(* PLC project EbN0扫描捕获_1度波束扫描及自跟踪优化 - 副本.project, CODESYS CODESYS V3.5 SP18 *)
(* stored: creationDateTime 2026-09-07T15:59:43.6480034, modificationDateTime 2026-09-07T15:13:02.4001786 *)

TYPE AxisCrtlStruct :
STRUCT
	iMode:INT;                     //方位运动模式   
	//bEnable :BOOL;                 //方位使能      
	rPosCmd :REAL;                 //方位位置命令    
	rVelCmd :REAL;                 //方位速度指令  
	rPIDCmdVel:LREAL;                //PID下发速度
	rPIDCmdPos:LREAL;				//PID目标位置
	bPIDEnable :BOOL;              //方位PID使能  
	bStartAutoTrack :BOOL;			//自跟踪使能
	rChanU:REAL;					//自跟踪采用的跟踪接收机误差电压
	
	rP:REAL:=1.0;                        //  P 
	rI:REAL:=0;                         //  I 
	rD:REAL:=0;                         //  D 
	rPIDThre:INT:=1;                   //积分阈值
	
	rP_AutoTrack:REAL:=3.0;          //自跟踪P
	rI_AutoTrack:REAL:=0.02;         //自跟踪I
	
	rAcceleration :REAL:=3;             //加速度
	rDeceleration :REAL:=3;       		//减速度
	rJogVel:LREAL:=2;					//点动速度 
	Pos_Vel:REAL:=4;					//位置模式速度
	rPos_Limit:LREAL;					//最大位置限制
	rVel_Limit:LREAL:=3;				//最大速度限制
	    
	rSoft_limit_Postive:REAL;
	rSoft_limit_Negative:REAL;			//正负软限位
	rLimitionNegative:LREAL;			//起始减速负限位
	rLimitionPositive:LREAL;			//起始减速正限位
	
END_STRUCT
END_TYPE

TYPE AxisStatus :
STRUCT
	Valid:BOOL;            //轴可用
	Busy:BOOL;             //轴工作中
	Error:BOOL;            //轴报错
	ErrorID:UINT;          //错误码
	ErrorStop:BOOL;        //轴错误停止
	Disabled:BOOL;         //轴下使能
	Stopping:BOOL;         //轴挂机或停止中
	Homing:BOOL;           //轴回原点
	Standstill:BOOL;       //轴待命
	DiscreteMotion:BOOL;   //轴离散运动
	ContinuousMotion:BOOL; //轴连续运动
	bServo_Enable:BOOL;		//轴使能状态
	bBrake:BOOL;			//轴抱闸状态
	Moving:BOOL;           //轴运动中
END_STRUCT
END_TYPE

TYPE AxisVisible :
STRUCT
	
	
	bJog_Forward:BOOL :=FALSE;
	bJog_Backward:BOOL :=FALSE;
	bVel_Run:BOOL:=FALSE;
	bPos_Run:BOOL:=FALSE;
	

	
	//JogB:BOOL;//点动指示灯
	//JogF:BOOL;
	bEnable:BOOL;//使能指示灯
	bUnable:BOOL;//下使能指示灯
	bLocalCtrl:BOOL;//本控指示灯
	bRemoteCtrl:BOOL;//远控指示灯
	//bJogLight:BOOL;//点动指示灯
	bStop:BOOL;//停止指示灯
	bmoveLight:BOOL;
	//bMovePos:BOOL;//速度运行指示灯
	//bMoveVel:BOOL;//位置运行指示灯
	bErrLight:BOOL;//报错提示灯
	//bExitPosLight:BOOL;//退限位模式指示灯
	//bPosLimLight:BOOL;//撞限位指示灯
	
	
	rLocalPosCmd:REAL;//本控位置命令
	rLocalVelCmd:REAL;//本控速度命令
	//rVelStep:REAL;//速度步距
	//rPosStep:REAL;//位置步距
END_STRUCT
END_TYPE

{attribute 'qualified_only'}
{attribute 'strict'}
TYPE MODES :
(
	powerOff:=0,          //下电
	powerOn := 1,         //上电
	positionMode:=2,      //位置模式
	velocityMode:=3,      //手动速度模式
	programBootMode:=4,   //程序引导模式
	reset:=6,             //轴错误复位
	halt:=7,              //停止
	stop:=8,             //挂机
	jog:=9 ,             //退限位模式
	edge:=10,            //
	test1:=11
);
END_TYPE

TYPE Word2Bit : UNION
  Apart_Word : WORD;
  Apart_Byte : ARRAY[1..2] OF BYTE;
  Apart_Real : REAL;  (* Apart_Bit:ARRAY[1..32]OF BIT; *)
  Apart_Int : INT;
END_UNION;
END_TYPE

TYPE Dword2Bit : UNION
  Apart_Dword : DWORD;
  Apart_Word : ARRAY[1..2] OF WORD;
  Apart_Byte : ARRAY[1..4] OF BYTE;
  Apart_Real : REAL;  (* Apart_Bit:ARRAY[1..32]OF BIT; *)
  Apart_Int : INT;
END_UNION;
END_TYPE

TYPE float2bit : UNION
  Apart_ulint : ULINT;
  Apart_dword : ARRAY[1..2] OF DWORD;
  Apart_word : ARRAY[1..4] OF WORD;
  Apart_byte : ARRAY[1..8] OF BYTE;
  Apart_real : ARRAY[1..2] OF REAL;  (* Apart_bit:ARRAY[1..64]OF Util.BIT_AS_DWORD; *)
  Apart_int : ARRAY[1..4] OF INT;
END_UNION;
END_TYPE

TYPE UnionLREAL_WORD : UNION
  lrealValue : LREAL;
  words : ARRAY[1..4] OF WORD;
END_UNION;
END_TYPE

TYPE Time2Word : UNION
  uliData : ULINT;
  wWords : ARRAY[1..4] OF WORD;
  lrReal : LREAL;
  arReal : ARRAY[0..1] OF REAL;
END_UNION;
END_TYPE

PROGRAM PLC_PRG
VAR
	a : DINT;
	b : REAL;
END_VAR

                    a := REAL_TO_DINT(b * 524288 / 360);
                  
END_PROGRAM

PROGRAM TimeCase
VAR
	stUTC_Timestamp :SYSTIME ;
	stSYS_Timestamp :ULINT ;
	stGNSS_Timestap :ULINT;
    Result : RTS_IEC_RESULT;
	Uptriger:Standard.R_TRIG;
	Triger AT %IX0.0:BOOL;
	Feed AT %QX0.0:BOOL;	
	TON_F: TON;
	dDelPTime: DINT;
	max_DelPTime:DINT :=0; 
	min_DelPTime: DINT :=-999999;
	iCount: INT;
	dtNow: DATE_AND_TIME;
	dtGNSS: DATE_AND_TIME;
	dtLastGNSS: ULINT;
	iDiffETime: DINT;
	DelPTime: DINT;
	
END_VAR

                    //计算时间误差序列
Result := SysTimeRtcHighResGet(stUTC_Timestamp);        
stSYS_Timestamp := TO_ULINT(stUTC_Timestamp);           // ULINT，获取本地时间
dtNow := TO_DT(stUTC_Timestamp / 1000); 		        // 转换为DATE_AND_TIME类型

Uptriger(CLK:=Triger);                                  //检测PPS上升沿
IF Uptriger.Q THEN                                      //上升沿触发后，GPRMC解析，DO0上升沿输出（电平24V）
	Feed:=TRUE;	
	dtGNSS := TO_DT(GVL.stGNSS_Timestap / 1000); 	    // 拿到串口时间数据			                                     
	iDiffETime:=ULINT_TO_DINT(GVL.stGNSS_Timestap-dtLastGNSS);  
	dtLastGNSS:=GVL.stGNSS_Timestap;                    //缓存上一周期时间戳（ms)  
	dDelPTime:=ULINT_TO_DINT(GVL.stGNSS_Timestap - stSYS_Timestamp);       //计算误差	              
	IF iDiffETime = 1000 THEN                           //确保时间更新步进1S
		IF dDelPTime < 0 THEN                           //更新最小值
			IF dDelPTime < min_DelPTime THEN
				min_DelPTime:=dDelPTime;
				DelPTime:=min_DelPTime;                 
			END_IF		
		ELSE                                            //更新最大值
			IF dDelPTime > max_DelPTime THEN
				max_DelPTime:=dDelPTime;
				DelPTime:=max_DelPTime;
			END_IF
		END_IF	
	END_IF				    						
	iCount:=iCount+1;
	IF iCount >= 60 THEN                                //一分钟校一次时间
		GVL.dDelTime:=DelPTime;
		max_DelPTime:=0;
		min_DelPTime:=0;	
		iCount:=0;
	END_IF
	
END_IF
TON_F(IN:=Feed, PT:=T#100MS, Q=>,ET=>);                 //脉宽200ms（测试时延，为了在示波器看波形）
IF TON_F.Q THEN
	Feed:=FALSE;		
END_IF
                  
END_PROGRAM

FUNCTION_BLOCK PID
VAR_INPUT
    rTarget : REAL;       (* 设定值 *)
    rFeedback : REAL;       (* 反馈值 *)
	rPosLimPositive:LREAL;//位置正限位
	rPosLimNegative:LREAL;//位置反限位
	rKp:REAL;     //比例增益
	rKi:REAL;     //积分增益
	rKd:REAL;     //微分增益
	iThreshold:INT;//积分项开启的位置阈值
	bPIDEnable:BOOL:=TRUE;//PID使能
	rVelLim:LREAL;//速度限制
END_VAR
VAR_OUTPUT
    rPIDOutput : LREAL:=0;         //带方向的输出速度
	rPIDtrace : LREAL:=0;         //带方向的输出速度
END_VAR
VAR
	//rPIDOutPut: REAL:=0.0;
	rLastError: LREAL:=0.0;(*上一次误差*)
	rErrorNow:LREAL:=0.0;(*当前误差*)
    rIntegralNew : LREAL := 0.0; (* 积分项 *)
    rDerivativeNew : LREAL := 0.0; (* 微分项 *)
	rDelta: LREAL;(*增量*)
	rProportionNew: LREAL;
	
	//iAzPIDEnable: INT;
END_VAR

                    
IF (bPIDEnable>0) THEN //如果PID使能
	IF rTarget=rFeedback THEN
		rPIDOutput:=0;	
	ELSE
	
		rErrorNow:=rTarget-rFeedback;//计算当前误差 en
		rProportionNew:=rErrorNow;//比例项
		//积分项
		IF rFeedback>rPosLimNegative AND rFeedback<rPosLimPositive THEN //若在软限位之内，工作时开启积分项
			IF (ABS(rTarget-rFeedback)<iThreshold) THEN//位置差小于积分阈值
				rIntegralNew:= rIntegralNew+rErrorNow; //积分项
			ELSE
				rIntegralNew:=0;
			END_IF;
		ELSE //不在软限位范围内,则积分项为0
			rIntegralNew:=0;
		END_IF

		//PID输出
		rPIDOutPut:=rKp*rProportionNew+rKi*rIntegralNew;
		rPIDtrace:=rKp*rProportionNew+rKi*rIntegralNew;


		//PID限速
		
			IF rPIDOutput<(-rVelLim) THEN
				rPIDOutput:=-rVelLim;
			ELSIF rPIDOutput>rVelLim THEN
				rPIDOutput:=rVelLim;
			END_IF
		
		
		IF rFeedback>rPosLimPositive AND rPIDOutput>0 THEN 
			rPIDOutput:=0;
		END_IF
		IF rFeedback<rPosLimNegative AND rPIDOutput<0 THEN
			rPIDOutput:=0;
		END_IF
		
		rLastError:=rErrorNow;//将当前误差赋值给上一次误差
		
	END_IF
ELSE//非使能清零PID各项
	rProportionNew:=0.0;
	rIntegralNew:=0.0;
	rPIDOutput:=0.0;
END_IF










                  
END_FUNCTION_BLOCK

PROGRAM TimeAdd
VAR
	icount : INT;
	iSecondLast:INT;
END_VAR

                    // 监测时统串口状态，时间插值
IF iSecondLast <> GPRMC_1.iSecond THEN
	icount := 0;
ELSE
	icount := icount + 1;
END_IF
iSecondLast := GPRMC_1.iSecond;

IF icount > 2000 THEN
	icount := 0;
END_IF
                  
END_PROGRAM

PROGRAM GPRMC
VAR
	com_init:gcan.FB_Com_Init;      		//gcan.FB_Com_Init为串口初始化功能块，可设定串口端口号，串口波特率等参数
	com_read:gcan.FB_Com_Read ;				//gcan.FB_Com_Read为串口接收功能块，用于通过接收串口发送给PLC的数据
	com_write:gcan.FB_Com_Write ;			//gcan.FB_Com_Write为串口发送功能块，用于发送串口数据
	m_uiError:UINT;							//用于承接功能块中报错引脚错误信息的变量
	m_out:BOOL;								//用于承接功能块中完成标志引脚数据的变量
	isFirst:BOOL:=TRUE;						//用于判断初始化只执行一次的逻辑
	mPort:BYTE;								//程序中用作设定串口端口号
	recSize:UINT;							//接收数据长度，单位：字节
	recBuf:ARRAY[0..100] OF BYTE;			//用于存放接收到的串口数据的数组
	sum_i:INT;
	checksum:BYTE;
	iYear: INT;
	iMonth: INT;
	iDay: INT;
	iHour: INT;
	iMinute: INT;
	iSecond: INT;
	strDateTimeNow : STRING;
	gnssTimestamp: ULINT;
	high4: BYTE;
	low4: BYTE;
END_VAR

                    ////////////////////////////////////////////////////////////////////////////////////////
//串口接收GPRMC报文解析
//日期：2024/08/25
//版本：V1.1
/////////////////////////////////////////////////////////////////////////////////////////

mPort:=1;								//串口端口号设定，GCAN-PLC-400、GCAN-PLC-510、GCAN-PLC-511，1为232，2为485
										//GCAN-PLC-324、GCAN-PLC-326，1为第一路485，2为第2路485
IF isFirst THEN
	com_init(							//串口初始化功能块
	EN_IN:=TRUE,						//串口初始化功能块使能
	xEnable:=TRUE,						//串口功能使能
	bPort:=mPort,						//串口端口号设定
	uiBaudrate:=115200,					//串口波特率设定
	bParity:=0,							//串口奇偶校验设定，0为无校验，1为奇校验，2为偶检验
	bDatabits:=8,						//数据位设定
	bStopbits:=1,						//停止位设定
	EN_OUT=>m_out,						//串口初始化功能块执行完成标志位
	uiError=>m_uiError);				//串口初始化功能块执行错误信息
	isfirst:=FALSE;						//执行一次初始化后关闭IF的条件使其之后进入ELSE程序段运行

ELSE
	
		com_read(						//串口读取功能块
		EN_in:=TRUE,					//读取功能块使能，为TRUE执行读取
		bPort:=mPort,					//串口端口号设定
		p_brxdata:=ADR(recBuf),			//读取到的串口数据引脚为指针类型，使用ADR()指向自建数组将数据存放到数组中
		uiMaxsize:=100,					//设定最大读取长度
		EN_out=>m_out,					//串口读取功能块执行完成标志位******功能块执行完成不代表接收完成********
		uiRecSize=>recSize,				//串口接收数据长度，单位：字节，大于0时说明接收到数据可用于判断是否接收
		uierror=>m_uierror);			//串口读取功能块执行错误信息
										//从数组recBuf里取数据，解析出年、月、日、时、分、秒
		//有效判定(A)+和校验(hh),前 4bit和后 4bit的 16 进制数分别以 ASCII 码表示(0~9,A~F)，高位在前。
		IF 	recBuf[17] = 65 THEN
(*			checksum := 16#00;
			FOR sum_i:=1 TO 74 BY 1 DO
				checksum:= checksum XOR recBuf[sum_i];
			END_FOR
			high4 := (SHR(checksum, 4) AND 16#0F)+16#30;
			low4 := (checksum AND 16#0F)+16#30;
			IF recBuf[76]= high4 AND recBuf[77]= low4 THEN 
*)			IF recBuf[60] = 44 THEN // 航向角 x.x
				iYear:=BYTE_TO_INT(recBuf[65]-48)*10+BYTE_TO_INT(recBuf[66]-48)+2000;
				iMonth:=BYTE_TO_INT(recBuf[63]-48)*10+BYTE_TO_INT(recBuf[64]-48);
				iDay:=BYTE_TO_INT(recBuf[61]-48)*10+BYTE_TO_INT(recBuf[62]-48);
				iHour:=BYTE_TO_INT(recBuf[7]-48)*10+BYTE_TO_INT(recBuf[8]-48)+8;
				iMinute:=BYTE_TO_INT(recBuf[9]-48)*10+BYTE_TO_INT(recBuf[10]-48);
				iSecond:=BYTE_TO_INT(recBuf[11]-48)*10+BYTE_TO_INT(recBuf[12]-48);
			END_IF
			IF recBuf[61] = 44 THEN // 航向角 xx.x
				iYear:=BYTE_TO_INT(recBuf[66]-48)*10+BYTE_TO_INT(recBuf[67]-48)+2000;
				iMonth:=BYTE_TO_INT(recBuf[64]-48)*10+BYTE_TO_INT(recBuf[65]-48);
				iDay:=BYTE_TO_INT(recBuf[62]-48)*10+BYTE_TO_INT(recBuf[63]-48);
				iHour:=BYTE_TO_INT(recBuf[7]-48)*10+BYTE_TO_INT(recBuf[8]-48)+8;
				iMinute:=BYTE_TO_INT(recBuf[9]-48)*10+BYTE_TO_INT(recBuf[10]-48);
				iSecond:=BYTE_TO_INT(recBuf[11]-48)*10+BYTE_TO_INT(recBuf[12]-48);
			END_IF
			IF recBuf[62] = 44 THEN // 航向角 xxx.x
				iYear:=BYTE_TO_INT(recBuf[67]-48)*10+BYTE_TO_INT(recBuf[68]-48)+2000;
				iMonth:=BYTE_TO_INT(recBuf[65]-48)*10+BYTE_TO_INT(recBuf[66]-48);
				iDay:=BYTE_TO_INT(recBuf[63]-48)*10+BYTE_TO_INT(recBuf[64]-48);
				iHour:=BYTE_TO_INT(recBuf[7]-48)*10+BYTE_TO_INT(recBuf[8]-48)+8;
				iMinute:=BYTE_TO_INT(recBuf[9]-48)*10+BYTE_TO_INT(recBuf[10]-48);
				iSecond:=BYTE_TO_INT(recBuf[11]-48)*10+BYTE_TO_INT(recBuf[12]-48);
			END_IF
				// 计算时间戳		
				strDateTimeNow := CONCAT(STR1 := 'DT#', STR2 := INT_TO_STRING(iYear));
				strDateTimeNow := CONCAT(STR1 := strDateTimeNow, STR2 := '-');
				strDateTimeNow := CONCAT(STR1 := strDateTimeNow, STR2 := INT_TO_STRING(iMonth));
				strDateTimeNow := CONCAT(STR1 := strDateTimeNow, STR2 := '-');
				strDateTimeNow := CONCAT(STR1 := strDateTimeNow, STR2 := INT_TO_STRING(iDay));
				strDateTimeNow := CONCAT(STR1 := strDateTimeNow, STR2 := '-');
				strDateTimeNow := CONCAT(STR1 := strDateTimeNow, STR2 := INT_TO_STRING(iHour));
				strDateTimeNow := CONCAT(STR1 := strDateTimeNow, STR2 := ':');
				strDateTimeNow := CONCAT(STR1 := strDateTimeNow, STR2 := INT_TO_STRING(iMinute));
				strDateTimeNow := CONCAT(STR1 := strDateTimeNow, STR2 := ':');
				strDateTimeNow := CONCAT(STR1 := strDateTimeNow, STR2 := INT_TO_STRING(iSecond));
				gnssTimestamp := DT_TO_ULINT(TO_DT(strDateTimeNow)) * 1000;
				GVL.stGNSS_Timestap := gnssTimestamp;
			//END_IF
		END_IF
					


(*	IF recsize>0 THEN					//如果接收到串口数据
		
		com_write(						//串口发送功能块
		EN_IN:=TRUE,					//串口发送功能块使能，发送机制：当使能为TRUE时，PLC程序每周期运行到此处就执行一次发送
		bPort:=mPort,					//串口端口号设定
		p_bTxdata:=ADR(recbuf),			//将接收存放到数组中的数据发送出去******若发送其它数据，自建另一数组用于存放发送数据即可
		uiTxsize:=recsize,				//发送长度为接收到的数据长度******若发送其它长度，自行填写所需长度即可
		EN_OUT=>m_out,					//串口发送功能块执行完成标志位
		uierror=>m_uierror);			//串口发送功能块执行错误信息
			
	END_IF
*)	
END_IF
                  
END_PROGRAM

PROGRAM RealTimePosCal
VAR
	dtReal: DATE_AND_TIME;
	sRealTime:STRING;
	btestTimeInit:BOOL;
	AzCubicInter:threesimple2_1;//方位三次样条插值
	ElCubicInter:threesimple2_1;//俯仰三次样条插值
	iErrcode : INT;
	rInterAzPos:REAL;//方位轴插值位置
    rInterElPos:REAL;//俯仰轴插值位置
	
	rInterAzPostest:REAL;//方位轴插值位置
    rInterElPostest:REAL;//俯仰轴插值位置
	
	rPolyAzPos:REAL;//方位轴多项式位置
    rPolyElPos:REAL;//俯仰轴多项式位置
	AzPoly:Get_AZ;
	ElPoly:Get_AZ_1;
	
	dRTime:ULINT;//上位机外部时间 单位ns Unix时间戳，起点是1970-1-1 0:0:0
	dLastRTime:ULINT;
	icount : INT;
END_VAR

                    //GVL.dRealTime:= TimeCase.stSYS_Timestamp + GVL.dDelTime + 1000 + 56 ;// 矫正后的时间 单位毫秒
//GVL.dRealTime:= TimeCase.stSYS_Timestamp + GVL.dDelTime;// 矫正后的时间 单位毫秒

//直接从上位机拿数
dRTime := modbus_slave.UTC_New + 8 * 3600 * 1000;
IF dRTime <> dLastRTime THEN
	icount := 0;
ELSE 
	icount := icount + 1;
END_IF
dLastRTime:=dRTime;
IF not GVL.bTimeSwich THEN
	GVL.dRealTime:=GVL.stGNSS_Timestap + 10*timeadd.icount;
ELSE
	GVL.dRealTime:=dRTime + 10*icount;
END_IF
IF icount > 5000 THEN
	icount := 0;
END_IF
(*
GVL.dRealTime:=GVL.stGNSS_Timestap + 10*timeadd.icount;
*)
dtReal := TO_DT(GVL.dRealTime / 1000);
sRealTime := TO_STRING(dtReal);

IF Axis1Remote.iMode=4 AND Axis2Remote.iMode=4 THEN//若PTP时间锁定 且时间模式为PTP时间
		//三次样条插值

		//GVL.dRealTime:= TimeCase.stSYS_Timestamp + GVL.dDelTime + 1000 + 56; // 矫正后的时间 单位毫秒
		IF NOT GVL.bTimeSwich THEN
			GVL.dRealTime:=GVL.stGNSS_Timestap + 10*timeadd.icount;
		ELSE
			GVL.dRealTime:=dRTime + 10*icount;
		END_IF
		AzCubicInter(XModbusUL:=Modbus_Slave.aUTC_TIME,YModbus:=Modbus_Slave.aPosCmd_2,y0:=0,yn:=0,xt:=(ULINT_TO_LREAL(GVL.dRealTime) - 8 * 3600 *1000),sout=>rInterAzPos,ErrCode=>iErrcode);
		ElCubicInter(XModbusUL:=Modbus_Slave.aUTC_TIME,YModbus:=Modbus_Slave.aPosCmd_1,y0:=0,yn:=0,xt:=(ULINT_TO_LREAL(GVL.dRealTime) - 8 * 3600 *1000),sout=>rInterElPos,ErrCode=>iErrcode);
		IF iErrcode>0 THEN //模块内错误代码清0 外部维持
			Error_code:=iErrcode;
		END_IF
END_IF
(*
//IF Axis1Remote.iMode=4 AND Axis2Remote.iMode=4 AND Modbus_Slave.bIFPoly THEN//若PTP时间锁定 且时间模式为PTP时间
IF Modbus_Slave.bIFPoly THEN//若PTP时间锁定 且时间模式为PTP时间
		//多项式拟合

		//GVL.dRealTime:= TimeCase.stSYS_Timestamp + GVL.dDelTime + 1000 + 56; // 矫正后的时间 单位毫秒
		GVL.dRealTime:= GVL.stGNSS_Timestap +450; // 矫正后的时间 单位毫秒
	
		AzPoly(
		uliRealTime := (ULINT_TO_LREAL(GVL.dRealTime) - 8 * 3600 *1000),
		lrStartTime := Modbus_Slave.starttime,
		rNodeTime1 := Modbus_Slave.rNodeTime1_az,
		rNodeTime2 := Modbus_Slave.rNodeTime2_az,
		rNodeTime3 := Modbus_Slave.rNodeTime3_az,
		rNodeTime4 := Modbus_Slave.rNodeTime4_az,
		rNodeTime5 := Modbus_Slave.rNodeTime5_az,
		rEndTime := Modbus_Slave.rEndTime,
		lrFun1 := Modbus_Slave.lrFun1_az,
		lrFun2 := Modbus_Slave.lrFun2_az,
		lrFun3 := Modbus_Slave.lrFun3_az,
		lrFun4 := Modbus_Slave.lrFun4_az,
		lrFun5 := Modbus_Slave.lrFun5_az,
		lrFun6 := Modbus_Slave.lrFun6_az,
		lrFitResult => rPolyAzPos);
		
		ElPoly(
		uliRealTime := (ULINT_TO_LREAL(GVL.dRealTime) - 8 * 3600 *1000),
		lrStartTime := Modbus_Slave.starttime,
		rNodeTime1 := Modbus_Slave.rNodeTime1_el,
		rNodeTime2 := Modbus_Slave.rNodeTime2_el,
		rNodeTime3 := Modbus_Slave.rNodeTime3_el,
		rNodeTime4 := Modbus_Slave.rNodeTime4_el,
		rNodeTime5 := Modbus_Slave.rNodeTime5_el,
		rEndTime := Modbus_Slave.rEndTime,
		lrFun1 := Modbus_Slave.lrFun1_el,
		lrFun2 := Modbus_Slave.lrFun2_el,
		lrFun3 := Modbus_Slave.lrFun3_el,
		lrFun4 := Modbus_Slave.lrFun4_el,
		lrFun5 := Modbus_Slave.lrFun5_el,
		lrFun6 := Modbus_Slave.lrFun6_el,
		lrFitResult => rPolyElPos);
		
		rInterAzPos := rPolyAzPos * (-1);
		rInterElPos := rPolyElPos + 90;
END_IF
*)
                  
END_PROGRAM

PROGRAM Modbus_Slave
VAR
	modTcpSlaveInit:gcan.FB_ModbusTCP_Slave_Init;	//gcan.FB_ModbusTCP_Slave_Init为Modbus TCP Slave初始化功能块
	modTcpSlaveCtrl:gcan.FB_ModbusTCP_Slave_Ctrl;	//gcan.FB_ModbusTCP_Slave_Init为Modbus TCP Slave执行功能块
	eout: BOOL;										//用于承接功能块中完成标志引脚数据的变量
	iSocket: INT;									//用于存放自身socket
	uiErr: UINT;									//用于承接功能块中报错引脚错误信息的变量
	isInit: BOOL:=FALSE;							//用于初始化执行一次的逻辑变量
	arClient:ARRAY[0..10] OF INT;					//用于存放Client即主站的socket
	
	arDo_data:ARRAY[0..654] OF BOOL;					//用于存放线圈的数据
	arDi_data:ARRAY[0..79] OF BOOL;					//用于存放离散型数据
	//arReg_data:ARRAY[0..10] OF INT;					//用于存放保持型寄存器的数据
	//arAi_data:ARRAY[0..10] OF INT;					//用于存放输入型寄存器的数据
	modbusData	    AT %MW0		: ARRAY[0..654] OF WORD;//用于存放保持型寄存器的数据，接收的数据
	modbusInputRegs	AT %MW660	: ARRAY[0..79] OF WORD;//用于存放输入型寄存器的数据，上报的数据
	
	enCtr:BOOL:=FALSE;								//Modbus TCP Slave执行功能块使能变量

	Remote_time 	 	:LWORD;
	dif:ULINT;//时延
	iCount				:WORD;
	TypeList1 			:DWORD;
	UTC_Union: float2bit;
	CtrlBool: WORD_AS_BIT;
	bCommReset:BOOL;		//错误复位标识符
	iWatchDogTime:INT;
	
	Pos1_Union:float2bit;//远控处理数据结构体
	Pos2_Union:float2bit;
	Pos3_Union:float2bit;
	//轴1远控指令，俯仰
	iMode_1 			:INT;  			//轴1模式远控
	rPosCmd_1 		 	:REAL; 			//轴1位置指令远控
	rVelcmd_1 			:REAL; 			//轴1速度指令远控
	rP_1 				:REAL;    	//轴1P远控
	rI_1 			 	:REAL;      	//轴1I远控
	rD_1				:REAL;     	//轴1D远控
	rThreshold_1 	 	:INT:=1;		//轴1积分阈值远控
	rAcceleration_1  	:REAL;			//最大加速度
	rDeceleration_1  	:REAL;			//最大减速度	
	rVelLim_1	  	 	:REAL;			//最大速度
	
	//轴2远控指令，方位
    iMode_2  		 	:INT; 			//轴2模式远控
	rPosCmd_2 			:REAL; 			//轴2位置指令远控
	rVelcmd_2 			:REAL; 			//轴2速度指令远控
	rP_2 				:REAL;  		//轴2P远控
	rI_2 			 	:REAL;  		//轴2I远控
	rD_2 			 	:REAL;  		//轴2D远控
	rThreshold_2 		:INT;			//轴2积分阈值远控
	rAcceleration_2 	:REAL;			//最大加速度
	rDeceleration_2  	:REAL;			//最大减速度	
	rVelLim_2	  		:REAL;			//最大速度
	//轴3远控指令，方位
    iMode_3  		 	:INT; 			//轴2模式远控
	rPosCmd_3 			:REAL; 			//轴2位置指令远控
	rVelcmd_3 			:REAL; 			//轴2速度指令远控
	rP_3 				:REAL;  		//轴2P远控
	rI_3 			 	:REAL;  		//轴2I远控
	rD_3 			 	:REAL;  		//轴2D远控
	rThreshold_3 		:INT;			//轴2积分阈值远控
	rAcceleration_3 	:REAL;			//最大加速度
	rDeceleration_3  	:REAL;			//最大减速度	
	rVelLim_3	  		:REAL;			//最大速度
	
	//轨道时间结构体
	UTC_Orbit_Union:float2bit;
	UTC_Orbit_New:ULINT;
	UTC_Orbit_Last:ULINT;
	//拉偏变量
	TimeBias_Union:float2bit;
	Bias1_Union:float2bit;
	Bias2_Union:float2bit;
	Bias3_Union:float2bit;
	AcuElOffset:float2bit;
	rTimeBias:LREAL;
	rBias_1:LREAL;
	rBias_2:LREAL;
	rBias_3:LREAL;
	lrElOffset:LREAL;
	UTC_New:ULINT;
	UTC_Last:ULINT;
	aUTC_TIME:ARRAY [1..10] OF ULINT;  //用于三次样条插值的数据
	aPosCmd_1 :ARRAY [1..10] OF LREAL;//用于三次样条插值的数据
	aPosCmd_2 :ARRAY [1..10] OF LREAL;//用于三次样条插值的数据
	isave:INT;
	iCheck:INT;
	bPass:BOOL;//通过大小检测
	iclear:INT;
	
	uPTPTime_Union:float2bit;
	DI1_Union:Util.BIT_AS_WORD;	//上报位置结构体
	DI2_Union:Util.BIT_AS_WORD;
	DO1_Union:Util.BIT_AS_WORD;
	DO2_Union:Util.BIT_AS_WORD;
	DI1_word:WORD;
	DI2_word:WORD;
	DO1_word:WORD;
	DO2_word:WORD;
// 	
	PosSub1_Union:float2bit;
	PosSub2_Union:float2bit;
	PosSub3_Union:float2bit;
	BiasSub1_Union:float2bit;
	BiasSub2_Union:float2bit;
	BiasSub3_Union:float2bit;

	Chan_Union:Util.BIT_AS_WORD;
	Chan_word:WORD;
	
	ptptime:ULINT;
	
	rAzTheory:LREAL;
	rEltheory:LREAL;
	rAzTheory_Union:float2bit;
	rEltheory_Union:float2bit;
	
	
	MillisecondsTime: ULINT;
	
	// for time test
	DeltaTimeBetPC : ULINT;

	AGC_Value: REAL;

	// 方位轨道多项式变量
	starttime : LREAL ;
	rNodeTime1_az : LREAL;
	rNodeTime2_az : LREAL;
	rNodeTime3_az : LREAL;
    rNodeTime4_az : LREAL;
    rNodeTime5_az : LREAL;
	rEndTime : LREAL;
	
	lrFun1_az : ARRAY[0..10] OF LREAL;
    lrFun2_az : ARRAY[0..10] OF LREAL;
    lrFun3_az : ARRAY[0..10] OF LREAL;
    lrFun4_az : ARRAY[0..10] OF LREAL;
	lrFun5_az : ARRAY[0..10] OF LREAL;
    lrFun6_az : ARRAY[0..10] OF LREAL;

    unionFun1_az : ARRAY[0..10] OF UnionLREAL_WORD;
    unionFun2_az : ARRAY[0..10] OF UnionLREAL_WORD;
    unionFun3_az : ARRAY[0..10] OF UnionLREAL_WORD;
    unionFun4_az : ARRAY[0..10] OF UnionLREAL_WORD;
    unionFun5_az : ARRAY[0..10] OF UnionLREAL_WORD;
    unionFun6_az : ARRAY[0..10] OF UnionLREAL_WORD;
	
	unionStartTime: UnionLREAL_WORD;
	
    unionNodeTime1_az : UnionLREAL_WORD;
    unionNodeTime2_az : UnionLREAL_WORD;
    unionNodeTime3_az : UnionLREAL_WORD;
    unionNodeTime4_az : UnionLREAL_WORD;
    unionNodeTime5_az : UnionLREAL_WORD;
    unionEndTime : UnionLREAL_WORD;
	
	// 俯仰轨道多项式变量
	rNodeTime1_el : REAL;
	rNodeTime2_el : REAL;
	rNodeTime3_el : REAL;
    rNodeTime4_el : REAL;
    rNodeTime5_el : REAL;
	lrFun1_el : ARRAY[0..10] OF LREAL;
    lrFun2_el : ARRAY[0..10] OF LREAL;
    lrFun3_el : ARRAY[0..10] OF LREAL;
    lrFun4_el : ARRAY[0..10] OF LREAL;
	lrFun5_el : ARRAY[0..10] OF LREAL;
    lrFun6_el : ARRAY[0..10] OF LREAL;
	unionFun1_el : ARRAY[0..10] OF UnionLREAL_WORD;
	unionFun2_el : ARRAY[0..10] OF UnionLREAL_WORD;
	unionFun3_el : ARRAY[0..10] OF UnionLREAL_WORD;
	unionFun4_el : ARRAY[0..10] OF UnionLREAL_WORD;
	unionFun5_el : ARRAY[0..10] OF UnionLREAL_WORD;
	unionFun6_el : ARRAY[0..10] OF UnionLREAL_WORD;
	unionNodeTime1_el : UnionLREAL_WORD;
	unionNodeTime2_el : UnionLREAL_WORD;
	unionNodeTime3_el : UnionLREAL_WORD;
	unionNodeTime4_el : UnionLREAL_WORD;
	unionNodeTime5_el : UnionLREAL_WORD;
	unionSum:UnionLREAL_WORD;
	lrSum:LREAL;
	lrSumlocal:LREAL;
	i : INT;
	bNotFirst : BOOL; //
	bCheck : BOOL;
	bIFPoly: BOOL;//开启多项式拟合模式的标识，由上位机下发
	iCountPolyGet:INT;//计时接收多项式数组的模块
	uChangeTest:Time2Word;//变量转换测试
	iCountSum:INT;
	bSearch: BOOL;
	bStartTrackAcu : BOOL;
	
	//接收上位机下发位置模式速度
	rAzPosVel : REAL := 8;
	rElPosVel : REAL := 6;
	rTlPosVel : REAL := 8;
END_VAR

                    IF isInit=FALSE THEN							
	
	modtcpslaveinit(en_in:=TRUE,					//Modbus TCP Slave初始化功能块使能
	xenable:=TRUE,									//使能初始化功能
	iport:=502,										//开放端口号502
	en_out=>eout,									//Modbus TCP Slave初始化功能块执行完成
	isocket=>iSocket,								//创建的socket存入变量
	uierror=>uiErr);								//Modbus TCP Slave初始化功能块执行错误信息
	
	IF isocket>=0 AND uiErr=0 THEN					//成功创建socket且无错误，逻辑标志置位，下周期执行ELSE
		isInit:=TRUE;	
		
		enCtr:=FALSE;
		ELSE                                        //等待连接成功
		modtcpslaveinit(en_in:=0,xenable:=0);	
	END_IF
	
 
ELSE
	
	modtcpslavectrl(en_in:=enCtr,					//Modbus TCP Slave执行功能块使能
	xenable:=TRUE,									//Modbus TCP Slave执行功能使能
	isocket:=isocket,								//输入创建的socket
	dwatchdogtime:=2000,							//看门狗时间
	p_clientsocket:=ADR(arClient),					//将连接进来的socket存放到数组
	imaxclientcount:=10,							//设置最大连接数量
	uido_number:=10,uido_startaddr:=0,pdo_data:=ADR(ardo_data),		//uido_number设定线圈个数，uido_startaddr设定线圈起始地址，数据存放在ardo_data数组
	uidi_number:=10,uidi_startaddr:=0,pdi_data:=ADR(ardi_data),		//uidi_number设定离散型数据个数，uidi_startaddr设定离散型数据起始地址，数据存放在ardi_data数组
	uireg_number:=655,uireg_startaddr:=0,preg_data:=ADR(modbusData), //uireg_number设定保持型寄存器个数，uireg_startaddr设定保持型寄存器起始地址，数据存放在arreg_data数组
	uiai_number:=79,uiai_startaddr:=0,pai_data:=ADR(modbusInputRegs),//uiai_number设定输入型寄存器个数，uiai_startaddr设定输入型寄存器起始地址，数据存放在arai_data数组
	en_out=>eout,									//Modbus TCP Slave执行功能块执行完成
	uierror=>uierr);								//Modbus TCP Slave执行功能块执行错误信息
	enctr:=TRUE;
	IF uierr <>0 THEN                               //如果从站报错，则重新连接从站
		modtcpslaveinit(en_in:=0,xenable:=0);	
		isInit:=0;
	END_IF
	//iMode:  0 下电  1 上电  2 速度模式  3 停止  4 位置模式  5 继续运行
	//方位轴指令
(*
	Az_ctrl.iMode:=WORD_TO_INT(modbusData[0]);
	AZ_ctrl.rTarVel:=WORD_TO_REAL(modbusData[1]);
	AZ_ctrl.rTarPos:=WORD_TO_REAL(modbusData[2])*-1.0;
	
	//俯仰轴指令
	El_ctrl.iMode:=WORD_TO_INT(modbusData[10]);
	El_ctrl.rTarVel:=WORD_TO_REAL(modbusData[11]);
	El_ctrl.rTarPos:=WORD_TO_REAL(modbusData[12])+90.0;
	*)
	
	// modbus下发数据
	UTC_Union.Apart_word[1]:=modbusData[3];
	UTC_Union.Apart_word[2]:=modbusData[2];
	UTC_Union.Apart_word[3]:=modbusData[1];
	UTC_Union.Apart_word[4]:=modbusData[0];
	UTC_New:=UTC_Union.Apart_ulint;
	DeltaTimeBetPC := UTC_New - TO_ULINT(GVL.dRealTime);
	CtrlBool(W:=modbusData[7],
			B14=>bCommReset,
			B13=>Axis2Remote.bPIDEnable,
			B12=>Axis1Remote.bPIDEnable,
			B11=>Axis3Remote.bPIDEnable,
			B10=>bStartTrackAcu,
			B07=>bIFPoly,
			B06=>bSearch, //十字搜索开启标识
			);
	//方位轴指令
	iMode_2:=WORD_TO_INT(modbusData[8]);
	Pos2_Union.Apart_word[2]:=modbusData[9];
	Pos2_Union.Apart_word[1]:=modbusData[10];
	rPosCmd_2:=DINT_TO_LREAL( DWORD_TO_DINT( Pos2_Union.Apart_dword[1]))/100000*-1;
	rVelcmd_2:=DINT_TO_LREAL( WORD_TO_INT(modbusData[11]))/1000*-1;
	rP_2:=INT_TO_LREAL(WORD_TO_INT(modbusData[12]))/1000;
	rI_2:=INT_TO_LREAL(WORD_TO_INT(modbusData[13]))/1000;
	rD_2:=INT_TO_LREAL(WORD_TO_INT(modbusData[14]))/1000;
	rThreshold_2:=WORD_TO_INT(modbusData[15])/1000;
	rAcceleration_2:=INT_TO_LREAL(WORD_TO_INT(modbusData[16]))/1000;
	rDeceleration_2:=INT_TO_LREAL(WORD_TO_INT(modbusData[17]))/1000;
	rVelLim_2:=INT_TO_LREAL(WORD_TO_INT(modbusData[18]))/1000;
	
	//俯仰轴指令
	iMode_1:=WORD_TO_INT(modbusData[19]);
	Pos1_Union.Apart_word[2]:=modbusData[20];
	Pos1_Union.Apart_word[1]:=modbusData[21];
	rPosCmd_1:=DINT_TO_LREAL( DWORD_TO_DINT( Pos1_Union.Apart_dword[1]))/100000+90;
	rVelcmd_1:=DINT_TO_LREAL( WORD_TO_INT(modbusData[22]))/1000;
	rP_1:=INT_TO_LREAL(WORD_TO_INT(modbusData[23]))/1000;
	rI_1:=INT_TO_LREAL(WORD_TO_INT(modbusData[24]))/1000;
	rD_1:=INT_TO_LREAL(WORD_TO_INT(modbusData[25]))/1000;
	rThreshold_1:=WORD_TO_INT(modbusData[26])/1000;
	rAcceleration_1:=INT_TO_LREAL(WORD_TO_INT(modbusData[27]))/1000;
	rDeceleration_1:=INT_TO_LREAL(WORD_TO_INT(modbusData[28]))/1000;
	rVelLim_1:=INT_TO_LREAL(WORD_TO_INT(modbusData[29]))/1000;
	
	//倾斜轴指令
	iMode_3:=WORD_TO_INT(modbusData[30]);
	Pos3_Union.Apart_word[2]:=modbusData[31];
	Pos3_Union.Apart_word[1]:=modbusData[32];
	rPosCmd_3:=DINT_TO_LREAL( DWORD_TO_DINT( Pos3_Union.Apart_dword[1]))/100000*-1;
	rVelcmd_3:=DINT_TO_LREAL( WORD_TO_INT(modbusData[33]))/1000*-1;
	rP_3:=INT_TO_LREAL(WORD_TO_INT(modbusData[34]))/1000;
	rI_3:=INT_TO_LREAL(WORD_TO_INT(modbusData[35]))/1000;
	rD_3:=INT_TO_LREAL(WORD_TO_INT(modbusData[36]))/1000;
	rThreshold_3:=WORD_TO_INT(modbusData[37])/1000;
	rAcceleration_3:=INT_TO_LREAL(WORD_TO_INT(modbusData[38]))/1000;
	rDeceleration_3:=INT_TO_LREAL(WORD_TO_INT(modbusData[39]))/1000;
	
	
	//AGC锁定门限
	AGC_Value:=(WORD_TO_UDINT(modbusData[43])/100.0);
	GVL.Chanthreshold:=AGC_Value;
	
	//轨道时间
	UTC_Orbit_Union.Apart_word[1]:=modbusData[48];
	UTC_Orbit_Union.Apart_word[2]:=modbusData[47];
	UTC_Orbit_Union.Apart_word[3]:=modbusData[46];
	UTC_Orbit_Union.Apart_word[4]:=modbusData[45];
	UTC_Orbit_New:=UTC_Orbit_Union.Apart_ulint;
	//时间拉偏
	TimeBias_Union.Apart_word[1]:=modbusData[50];
	TimeBias_Union.Apart_word[2]:=modbusData[49];
	rTimeBias:=DINT_TO_LREAL( DWORD_TO_DINT( TimeBias_Union.Apart_dword[1]))/100000.0; //单位为秒
	IF rTimeBias>0.4 THEN//时间偏置最大限制 正负0.4秒
		rTimeBias:=0.4;
	ELSIF rTimeBias<-0.4 THEN
		rTimeBias:=-0.4;
	END_IF
	rTimeBias:=rTimeBias*1000000000;//秒转纳秒
	//两轴拉偏
	Bias2_Union.Apart_word[1]:=modbusData[52];
	Bias2_Union.Apart_word[2]:=modbusData[51];
	rBias_2:=DINT_TO_LREAL( DWORD_TO_DINT( Bias2_Union.Apart_dword[1]))/100000.0*(-1);
	
	Bias1_Union.Apart_word[1]:=modbusData[54];
	Bias1_Union.Apart_word[2]:=modbusData[53];
	rBias_1:=DINT_TO_LREAL( DWORD_TO_DINT( Bias1_Union.Apart_dword[1]))/100000.0;
	
	//俯仰零值
	AcuElOffset.Apart_word[1]:=modbusData[58];
	AcuElOffset.Apart_word[2]:=modbusData[57];
	lrElOffset:=DINT_TO_LREAL( DWORD_TO_DINT( AcuElOffset.Apart_dword[1]))/100000.0;
	//存储modbus时间序列和位置命令序列
	//IF UTC_New<>UTC_Last THEN //命令刷新，则更新序列
	
	
	//接受位置模式速度下发
	rAzPosVel:=INT_TO_LREAL(WORD_TO_INT(modbusData[61]))/1000.0;
	rElPosVel:=INT_TO_LREAL(WORD_TO_INT(modbusData[62]))/1000.0;
	rTlPosVel:=INT_TO_LREAL(WORD_TO_INT(modbusData[63]))/1000.0;
	
	IF rAzPosVel <= 16.0 THEN
		GVL.Axis2Remote.Pos_Vel := rAzPosVel;
	ELSE
		GVL.Axis2Remote.Pos_Vel := 16;
	END_IF
	
	IF rElPosVel <= 11.0 THEN
		GVL.Axis1Remote.Pos_Vel := rElPosVel;
	ELSE
		GVL.Axis1Remote.Pos_Vel := 11;
	END_IF
	
	IF rTlPosVel <= 8.0 THEN
		GVL.Axis3Remote.Pos_Vel := rTlPosVel;
	ELSE
		GVL.Axis3Remote.Pos_Vel := 8;
	END_IF
	
	FOR iCheck:=1 TO 10 DO
		IF UTC_Orbit_New>aUTC_TIME[iCheck] THEN
			bPass:=TRUE;
		ELSE
			bPass:=FALSE;
			EXIT;
		END_IF
	END_FOR
	IF bPass THEN //命令刷新，则更新序列
		FOR isave:=1 TO 9 DO
			aUTC_TIME[isave]:=aUTC_TIME[isave+1];
			aPosCmd_1[isave]:=aPosCmd_1[isave+1];
			aPosCmd_2[isave]:=aPosCmd_2[isave+1];
		END_FOR
		aUTC_TIME[10]:=UTC_Orbit_New;
		aPosCmd_1[10]:=rPosCmd_1;
		aPosCmd_2[10]:=rPosCmd_2;
	END_IF
	//若不是程引模式，则清空轨道时间数据
	IF Axis1Remote.iMode<>4 AND Axis2Remote.iMode<>4 THEN
		FOR iCheck:=1 TO 10 DO
			aUTC_TIME[iCheck]:=0;;
		END_FOR
	END_IF
	
	// modbus上报数据	
	IF icount<16#FFFF THEN
		icount:=icount+1;
	ELSE
		icount:=0;
	END_IF
	
	DI1_Union(B15:=SecurityCheck.bPrelimit_Positive_1,						//俯仰轴预限位--正 B15=0为未触发，B15=1为触发
			B14:=SecurityCheck.bFinallimit_1,								//俯仰轴终限位
			B13:=SecurityCheck.bPrelimit_Negative_1,						//俯仰轴预限位--负
			B12:=SecurityCheck.bFinallimit_1,								//俯仰位终限位
			B11:=SecurityCheck.bPrelimit_Positive_2,						//方位轴预限位--正
			B10:=SecurityCheck.bFinallimit_2,								//方位轴终限位
			B09:=SecurityCheck.bPrelimit_Negative_2,						//方位轴预限位--负
			B08:=SecurityCheck.bFinallimit_2,								//方位轴终限位
			B07:=FALSE,												//倾斜预限位--正
			B06:=FALSE,												//倾斜终限位--正
			B05:=FALSE,												//倾斜预限位--负
			B04:=FALSE,												//倾斜终限位--负
			B03:=FALSE,												//方位轴过零检测
			B02:=Axis2Status.bBrake,								//方位轴抱闸状态 0为解抱闸，1为抱闸
			B01:=Axis1Status.bBrake,								//俯仰轴抱闸状态
			B00:=Axis3Status.bBrake,								//倾斜轴抱闸状态
			W=>DI1_word	);
			
	DI2_Union(B15:=FALSE,								//
			B14:=FALSE,								//
			B13:=FALSE,
			B12:=FALSE,
			B11:=FALSE,
			B10:=FALSE,
			B09:=FALSE,
			B08:=FALSE,
			B07:=FALSE,
			B06:=FALSE,
			B05:=GVL.bError_Reset,											//错误复位符
			B04:=GVL.bLocalCtrl,											//本远控标识符
			B03:=FALSE,									//退限位标识符
			B02:=Axis2Remote.bPIDEnable,											//方位轴PID使能状态
			B01:=Axis1Remote.bPIDEnable,											//俯仰轴PID使能状态
			B00:=Axis3Remote.bPIDEnable,											//倾斜轴PID使能状态
			W=>DI2_word);
	DO1_Union(B15:=FALSE,								//中心体急停指示灯
			B14:=FALSE,							//声光报警		1为触发，0为未触发
			B13:=FALSE,							//爬梯急停指示灯 B13=1为亮 B13=0为灭
			B12:=FALSE,							//机柜蜂鸣器	B12=1为触发，B12=0为未触发
			B11:=FALSE,							//限位释放指示灯 同上 
			B10:=FALSE,						//本远控指示灯	B10=1为本控，B10=0为远控
			B09:=FALSE,							//系统状态指示灯 B09=1为异常，B09=0为正常	
			B08:=Axis2Status.bBrake,								//方位轴抱闸输出 B08=1为抱闸输出 B08=1为解抱闸输出
			B07:=Axis1Status.bBrake,								//俯仰轴抱闸输出 同上
			B06:=Axis3Status.bBrake,								//倾斜轴抱闸输出 同上
			B05:=FALSE,										//方位风扇输出	B05=1为风扇运行，B05=0为风扇未运行
			B04:=FALSE,										//俯仰风扇输出	同上
			B03:=FALSE,										//倾斜风扇输出	同上
			B02:=Axis2Status.bServo_Enable,									//方位轴供电
			B01:=Axis1Status.bServo_Enable,									//俯仰轴供电
			B00:=Axis3Status.bServo_Enable,									//倾斜轴供电
			W=>DO1_word);
	DO2_Union(B15:=Axis2Status.bServo_Enable,//NOT(Axis1Status.Disabled),						//方位主电机使能状态
			B14:=Axis2Status.bServo_Enable,//NOT(Axis1Status.Disabled),							//方位从电机使能状态
			B13:=Axis1Status.bServo_Enable,//NOT(Axis2Status.Disabled),							//俯仰主电机使能状态		
			B12:=Axis1Status.bServo_Enable,//NOT(Axis2Status.Disabled),							//俯仰从电机使能状态
			B11:=Axis3Status.bServo_Enable,		//倾斜主电机使能状态
	 		B10:=Axis3Status.bServo_Enable,		//倾斜从电机使能状态
			B09:=Az_ctrl_1.bStop_2,			//方位轴主电机停止标识符
	 		B08:=Az_ctrl_1.bStop_2,					  //方位轴从电机停止标识符
	 		B07:=El_ctrl_1.bStop_1,		    //俯仰轴主电机停止标识符
			B06:=El_ctrl_1.bStop_1,				//俯仰轴从电机停止标识符
	 		B05:=Ti_ctrl_1.bStop_3,							//倾斜轴主电机停止标识符
			B04:=Ti_ctrl_1.bStop_3,							//倾斜轴从电机停止标识符
	 		B03:=0,
	 		B02:=0,
			B01:=0,
			B00:=0,
			W=>DO2_word	);
	
	//命令角与实际角偏差
	IF bLocalCtrl THEN
		IF  Axis1Local.iMode=4 THEN
			BiasSub1_Union.Apart_dword[1]:=DINT_TO_DWORD( REAL_TO_DINT((Axis1Local.rPosCmd-rFctPosReal_1)*100000.0));//读取位置
		ELSE
			BiasSub1_Union.Apart_dword[1]:=0;//读取位置
		END_IF
	ELSE
		IF Axis1Remote.iMode=2  THEN 
			BiasSub1_Union.Apart_dword[1]:=DINT_TO_DWORD( REAL_TO_DINT((Axis1Remote.rPosCmd-rFctPosReal_1)*100000.0));//读取位置
		ELSIF Axis1Remote.iMode=4 THEN
			BiasSub1_Union.Apart_dword[1]:=DINT_TO_DWORD( REAL_TO_DINT((RealTimePosCal.rInterElPos-rFctPosReal_1)*100000.0));//读取位置
		ELSE
			BiasSub1_Union.Apart_dword[1]:=0;//读取位置
		END_IF
	END_IF
	
	IF bLocalCtrl THEN
		IF Axis2Local.iMode=4 THEN
			BiasSub2_Union.Apart_dword[1]:=DINT_TO_DWORD( REAL_TO_DINT((Axis2Local.rPosCmd-rFctPosReal_2)*100000.0));//读取位置
		ELSE
			BiasSub2_Union.Apart_dword[1]:=0;//读取位置
		END_IF
	ELSE
		IF Axis2Remote.iMode=2 THEN
			BiasSub2_Union.Apart_dword[1]:=DINT_TO_DWORD( REAL_TO_DINT((Axis2Remote.rPosCmd-rFctPosReal_2)*100000.0));//读取位置
		ELSIF Axis2Remote.iMode=4 THEN
			BiasSub2_Union.Apart_dword[1]:=DINT_TO_DWORD( REAL_TO_DINT((rFctPosReal_2-RealTimePosCal.rInterAzPos)*100000.0));//读取位置
		ELSE
			BiasSub2_Union.Apart_dword[1]:=0;//读取位置
		END_IF
	END_IF
	
	IF bLocalCtrl THEN
		IF Axis3Local.iMode=4 THEN
			BiasSub3_Union.Apart_dword[1]:=DINT_TO_DWORD( REAL_TO_DINT((Axis3Local.rPosCmd-rFctPosReal_3)*100000.0));//读取位置
		ELSE
			BiasSub3_Union.Apart_dword[1]:=0;//读取位置
		END_IF
	ELSE
		IF Axis3Remote.iMode=2 THEN
			BiasSub3_Union.Apart_dword[1]:=DINT_TO_DWORD( REAL_TO_DINT((Axis3Remote.rPosCmd-rFctPosReal_3)*100000.0));//读取位置
		ELSIF Axis2Remote.iMode=4 THEN
			BiasSub3_Union.Apart_dword[1]:=DINT_TO_DWORD( REAL_TO_DINT((Axis3Remote.rPIDCmdPos-rFctPosReal_3)*100000.0));//读取位置
		ELSE
			BiasSub3_Union.Apart_dword[1]:=0;//读取位置
		END_IF
	END_IF
	
	// uPTPTime_Union.Apart_ulint:=TO_ULINT(GVL.dPTPCSTTime/1000000);
	uPTPTime_Union.Apart_ulint:=TO_ULINT((GVL.dRealTime - 8 * 3600 * 1000) * 1000000);
	modbusInputRegs[0]:=uPTPTime_Union.Apart_word[4];
	modbusInputRegs[1]:=uPTPTime_Union.Apart_word[3];
	modbusInputRegs[2]:=uPTPTime_Union.Apart_word[2];
	modbusInputRegs[3]:=uPTPTime_Union.Apart_word[1];
	modbusInputRegs[4]:=INT_TO_WORD( icount);
	modbusInputRegs[5]:=INT_TO_WORD(Error_code);//错误代码
	modbusInputRegs[6]:=DI1_word;
	modbusInputRegs[7]:=DI2_word;
	modbusInputRegs[8]:=DO1_word;
	modbusInputRegs[9]:=DO2_word;
	
	
	PosSub1_Union.Apart_dword[1]:=DINT_TO_DWORD( REAL_TO_DINT((rFctPosReal_1-90)*100000.0));//读取俯仰位置
	
	PosSub2_Union.Apart_dword[1]:=DINT_TO_DWORD( REAL_TO_DINT((rFctPosReal_2*-1)*100000.0));//读取方位位置
	
	PosSub3_Union.Apart_dword[1]:=DINT_TO_DWORD( REAL_TO_DINT((rFctPosReal_3*-1)*100000.0));//读取倾斜位置
	
	
	//方位轴状态
	modbusInputRegs[10]:=INT_TO_WORD(Axis2Remote.iMode);
	
	modbusInputRegs[13]:=PosSub2_Union.Apart_word[2];
	modbusInputRegs[14]:=PosSub2_Union.Apart_word[1];
	
	modbusInputRegs[17]:=INT_TO_WORD(REAL_TO_INT(rFctVelReal_2*1000.0));							//速度
	
	modbusInputRegs[19]:=REAL_TO_UINT(Axis2Remote.rP*1000);
	modbusInputRegs[20]:=REAL_TO_UINT(Axis2Remote.rI*1000);
	modbusInputRegs[21]:=REAL_TO_UINT(Axis2Remote.rD*1000);
	modbusInputRegs[22]:=REAL_TO_UINT(Axis2Remote.rPIDThre*1000);
	modbusInputRegs[23]:=INT_TO_WORD(REAL_TO_INT(securitycheck.rAzCurrent*100.0));
	
	
	//俯仰轴状态
	modbusInputRegs[27]:=INT_TO_WORD(Axis1Remote.iMode);
	
	modbusInputRegs[30]:=PosSub1_Union.Apart_word[2];
	modbusInputRegs[31]:=PosSub1_Union.Apart_word[1];
	
	modbusInputRegs[34]:=INT_TO_WORD(REAL_TO_INT(rFctVelReal_1*1000));							     //速度
	
	modbusInputRegs[36]:=REAL_TO_UINT(Axis1Remote.rP*1000);
	modbusInputRegs[37]:=REAL_TO_UINT(Axis1Remote.rI*1000);
	modbusInputRegs[38]:=REAL_TO_UINT(Axis1Remote.rD*1000);
	modbusInputRegs[39]:=REAL_TO_UINT(Axis1Remote.rPIDThre*1000);
	modbusInputRegs[40]:=INT_TO_WORD(REAL_TO_INT(securitycheck.rElCurrent*100.0));
	//倾斜轴状态
	modbusInputRegs[44]:=INT_TO_WORD(Axis3Remote.iMode);
	
	modbusInputRegs[47]:=PosSub3_Union.Apart_word[2];
	modbusInputRegs[48]:=PosSub3_Union.Apart_word[1];
	
	modbusInputRegs[51]:=INT_TO_WORD(REAL_TO_INT(rFctVelReal_3*1000.0));							//速度
	
	modbusInputRegs[53]:=REAL_TO_UINT(Axis3Remote.rP*1000);
	modbusInputRegs[54]:=REAL_TO_UINT(Axis3Remote.rI*1000);
	modbusInputRegs[55]:=REAL_TO_UINT(Axis3Remote.rD*1000);
	modbusInputRegs[56]:=REAL_TO_UINT(Axis3Remote.rPIDThre*1000);
	modbusInputRegs[57]:=INT_TO_WORD(REAL_TO_INT(securitycheck.rTlCurrent*100.0));
	//跟踪接收机预留
	
	modbusInputRegs[69]:=BiasSub2_Union.Apart_word[2];
	modbusInputRegs[70]:=BiasSub2_Union.Apart_word[1];
	modbusInputRegs[71]:=BiasSub1_Union.Apart_word[2];
	modbusInputRegs[72]:=BiasSub1_Union.Apart_word[1];
	modbusInputRegs[73]:=BiasSub3_Union.Apart_word[2];
	modbusInputRegs[74]:=BiasSub3_Union.Apart_word[1];
	//上报用于校相的方位俯仰轴理论值 （插值位置加当前拉偏位置）
	rAzTheory:=RealTimePosCal.rInterAzPos*(-1);
	rAzTheory_Union.Apart_dword[1]:=DINT_TO_DWORD(LREAL_TO_DINT(rAzTheory*100000.0));
	rEltheory:=RealTimePosCal.rInterElPos-90;
	rEltheory_Union.Apart_dword[1]:=DINT_TO_DWORD(LREAL_TO_DINT(rEltheory*100000.0));
	modbusInputRegs[75]:=rAzTheory_Union.Apart_word[2];
	modbusInputRegs[76]:=rAzTheory_Union.Apart_word[1];
	modbusInputRegs[77]:=rEltheory_Union.Apart_word[2];
	modbusInputRegs[78]:=rEltheory_Union.Apart_word[1];

	//跟踪接收机状态字上报
	Chan_Union(B15:=GVL.Chan1Lock,
			  B14:=GVL.Chan1Online,
			  B13:=GVL.Chan2Lock,
			  B12:=GVL.Chan2Online,
			  //B11:=GVL.bStartTrack,
			  B11:=Read_485.bEBN0Lock,
			  B10:=0,
			  B09:=0,
			  B08:=0,
			  B07:=0,
			  B06:=0,
			  B05:=0,
			  B04:=0,
			  B03:=0,
			  B02:=0,
			  B01:=0,
			  B00:=0,
			  w=>Chan_word);
			  (*
	IF GVL.Chan1AGC >= GVL.Chanthreshold THEN
		GVL.Chan1Lock:=TRUE;
	ELSE
		GVL.Chan1Lock:=FALSE;	
	END_IF
	*)
	//跟踪接收机数据上报
	// IF Ether_Cat.EL6022State=8 THEN
	IF TRUE THEN
			modbusInputRegs[59]:=Chan_word;
			modbusInputRegs[60]:=REAL_TO_WORD(GVL.Chan1AGC*1000);
			
	   IF GVL.Chan1Ua>0 THEN
			modbusInputRegs[61]:=REAL_TO_WORD(GVL.Chan1Ua*1000);
	   ELSE
			modbusInputRegs[61]:=(-1)*REAL_TO_WORD(65536-GVL.Chan1Ua*1000);	
			
	   END_IF
	   
	   IF GVL.Chan1Ue>0 THEN
			modbusInputRegs[62]:=REAL_TO_WORD(GVL.Chan1Ue*1000);
	   ELSE
			modbusInputRegs[62]:=(-1)*REAL_TO_WORD(65536-GVL.Chan1Ue*1000);	
			
	   END_IF
	   
			modbusInputRegs[63]:=REAL_TO_WORD(GVL.Chan2AGC*1000);
			modbusInputRegs[64]:=REAL_TO_WORD(GVL.Chan2Ua*1000);
			modbusInputRegs[65]:=REAL_TO_WORD(GVL.Chan2Ue*1000);
	ELSE
			modbusInputRegs[59]:=0;
			modbusInputRegs[60]:=0;
			modbusInputRegs[61]:=0;
			modbusInputRegs[62]:=0;
			modbusInputRegs[63]:=0;
			modbusInputRegs[64]:=0;
			modbusInputRegs[65]:=0;
	END_IF
	//多项式拟合数据接收
	//IF GVL.AzCtrl.iMode = 11 AND GVL.ElCtrl.iMode = 11 THEN
	iCountPolyGet:=iCountPolyGet+1;
	//IF iCountPolyGet=10 THEN
		iCountPolyGet:=0;
	IF TRUE THEN
		FOR i := 0 TO 10 DO
			unionFun1_az[i].words[1] := modbusdata[74 + 4 * i];
			unionFun1_az[i].words[2] := modbusdata[73 + 4 * i];
			unionFun1_az[i].words[3] := modbusdata[72 + 4 * i];
			unionFun1_az[i].words[4] := modbusdata[71 + 4 * i];
			lrFun1_az[i] := unionFun1_az[i].lrealValue;
			
			unionFun2_az[i].words[1] := modbusdata[118 + 4 * i];
			unionFun2_az[i].words[2] := modbusdata[117 + 4 * i];
			unionFun2_az[i].words[3] := modbusdata[116 + 4 * i];
			unionFun2_az[i].words[4] := modbusdata[115 + 4 * i];
			lrFun2_az[i] := unionFun2_az[i].lrealValue;
			
			unionFun3_az[i].words[1] := modbusdata[162 + 4 * i];
			unionFun3_az[i].words[2] := modbusdata[161 + 4 * i];
			unionFun3_az[i].words[3] := modbusdata[160 + 4 * i];
			unionFun3_az[i].words[4] := modbusdata[159 + 4 * i];
			lrFun3_az[i] := unionFun3_az[i].lrealValue;
			
			unionFun4_az[i].words[1] := modbusdata[206 + 4 * i];
			unionFun4_az[i].words[2] := modbusdata[205 + 4 * i];
			unionFun4_az[i].words[3] := modbusdata[204 + 4 * i];
			unionFun4_az[i].words[4] := modbusdata[203 + 4 * i];
			lrFun4_az[i] := unionFun4_az[i].lrealValue;
			
			unionFun5_az[i].words[1] := modbusdata[250 + 4 * i];
			unionFun5_az[i].words[2] := modbusdata[249 + 4 * i];
			unionFun5_az[i].words[3] := modbusdata[248 + 4 * i];
			unionFun5_az[i].words[4] := modbusdata[247 + 4 * i];
			lrFun5_az[i] := unionFun5_az[i].lrealValue;
			
			unionFun6_az[i].words[1] := modbusdata[294 + 4 * i];
			unionFun6_az[i].words[2] := modbusdata[293 + 4 * i];
			unionFun6_az[i].words[3] := modbusdata[292 + 4 * i];
			unionFun6_az[i].words[4] := modbusdata[291 + 4 * i];
			lrFun6_az[i] := unionFun6_az[i].lrealValue;
			
			unionFun3_el[i].words[1] := modbusdata[450 + 4 * i];
			unionFun3_el[i].words[2] := modbusdata[449 + 4 * i];
			unionFun3_el[i].words[3] := modbusdata[448 + 4 * i];
			unionFun3_el[i].words[4] := modbusdata[447 + 4 * i];
			lrFun3_el[i] := unionFun3_el[i].lrealValue;
			
			unionFun4_el[i].words[1] := modbusdata[494 + 4 * i];
			unionFun4_el[i].words[2] := modbusdata[493 + 4 * i];
			unionFun4_el[i].words[3] := modbusdata[492 + 4 * i];
			unionFun4_el[i].words[4] := modbusdata[491 + 4 * i];
			lrFun4_el[i] := unionFun4_el[i].lrealValue;
			
			unionFun1_el[i].words[1] := modbusdata[362 + 4 * i];
			unionFun1_el[i].words[2] := modbusdata[361 + 4 * i];
			unionFun1_el[i].words[3] := modbusdata[360 + 4 * i];
			unionFun1_el[i].words[4] := modbusdata[359 + 4 * i];
			lrFun1_el[i] := unionFun1_el[i].lrealValue;
			
			unionFun2_el[i].words[1] := modbusdata[406 + 4 * i];
			unionFun2_el[i].words[2] := modbusdata[405 + 4 * i];
			unionFun2_el[i].words[3] := modbusdata[404 + 4 * i];
			unionFun2_el[i].words[4] := modbusdata[403 + 4 * i];
			lrFun2_el[i] := unionFun2_el[i].lrealValue;
			
			unionFun5_el[i].words[1] := modbusdata[538 + 4 * i];
			unionFun5_el[i].words[2] := modbusdata[537 + 4 * i];
			unionFun5_el[i].words[3] := modbusdata[536 + 4 * i];
			unionFun5_el[i].words[4] := modbusdata[535 + 4 * i];
			lrFun5_el[i] := unionFun5_el[i].lrealValue;
			
			unionFun6_el[i].words[1] := modbusdata[582 + 4 * i];
			unionFun6_el[i].words[2] := modbusdata[581 + 4 * i];
			unionFun6_el[i].words[3] := modbusdata[580 + 4 * i];
			unionFun6_el[i].words[4] := modbusdata[579 + 4 * i];
			lrFun6_el[i] := unionFun6_el[i].lrealValue;
		END_FOR
		i:=0;
		unionNodeTime1_az.words[1] := modbusdata[338];
		unionNodeTime1_az.words[2] := modbusdata[337];
		unionNodeTime1_az.words[3] := modbusdata[336];
		unionNodeTime1_az.words[4] := modbusdata[335];
		rNodeTime1_az := unionNodeTime1_az.lrealValue;
		
		unionNodeTime2_az.words[1] := modbusdata[342];
		unionNodeTime2_az.words[2] := modbusdata[341];
		unionNodeTime2_az.words[3] := modbusdata[340];
		unionNodeTime2_az.words[4] := modbusdata[339];
		rNodeTime2_az := unionNodeTime2_az.lrealValue;
		
		unionNodeTime3_az.words[1] := modbusdata[346];
		unionNodeTime3_az.words[2] := modbusdata[345];
		unionNodeTime3_az.words[3] := modbusdata[344];
		unionNodeTime3_az.words[4] := modbusdata[343];
		rNodeTime3_az := unionNodeTime3_az.lrealValue;
		
		unionNodeTime4_az.words[1] := modbusdata[350];
		unionNodeTime4_az.words[2] := modbusdata[349];
		unionNodeTime4_az.words[3] := modbusdata[348];
		unionNodeTime4_az.words[4] := modbusdata[347];
		rNodeTime4_az := unionNodeTime4_az.lrealValue;
		
		unionNodeTime5_az.words[1] := modbusdata[354];
		unionNodeTime5_az.words[2] := modbusdata[353];
		unionNodeTime5_az.words[3] := modbusdata[352];
		unionNodeTime5_az.words[4] := modbusdata[351];
		rNodeTime5_az := unionNodeTime5_az.lrealValue;

		unionStartTime.words[1]:=modbusdata[646];
		unionStartTime.words[2]:=modbusdata[645];
		unionStartTime.words[3]:=modbusdata[644];
		unionStartTime.words[4]:=modbusdata[643];
		starttime:=unionStartTime.lrealValue;
		unionEndTime.words[1] := modbusdata[358];
		unionEndTime.words[2] := modbusdata[357];
		unionEndTime.words[3] := modbusdata[356];
		unionEndTime.words[4] := modbusdata[355];
		rEndTime := unionEndTime.lrealValue;
		
		//FOR i := 0 TO 5 DO
			
		//END_FOR
		
		unionNodeTime1_el.words[1] := modbusdata[626];
		unionNodeTime1_el.words[2] := modbusdata[625];
		unionNodeTime1_el.words[3] := modbusdata[624];
		unionNodeTime1_el.words[4] := modbusdata[623];
		rNodeTime1_el := unionNodeTime1_el.lrealValue;
		
		unionNodeTime2_el.words[1] := modbusdata[630];
		unionNodeTime2_el.words[2] := modbusdata[629];
		unionNodeTime2_el.words[3] := modbusdata[628];
		unionNodeTime2_el.words[4] := modbusdata[627];
		rNodeTime2_el := unionNodeTime2_el.lrealValue;
		
		unionNodeTime3_el.words[1] := modbusdata[634];
		unionNodeTime3_el.words[2] := modbusdata[633];
		unionNodeTime3_el.words[3] := modbusdata[632];
		unionNodeTime3_el.words[4] := modbusdata[631];
		rNodeTime3_el := unionNodeTime3_el.lrealValue;
		
		unionNodeTime4_el.words[1] := modbusdata[638];
		unionNodeTime4_el.words[2] := modbusdata[637];
		unionNodeTime4_el.words[3] := modbusdata[636];
		unionNodeTime4_el.words[4] := modbusdata[635];
		rNodeTime4_el := unionNodeTime4_el.lrealValue;
		
		unionNodeTime5_el.words[1] := modbusdata[642];
		unionNodeTime5_el.words[2] := modbusdata[641];
		unionNodeTime5_el.words[3] := modbusdata[640];
		unionNodeTime5_el.words[4] := modbusdata[639];
		rNodeTime5_el := unionNodeTime5_el.lrealValue;
		
		(*
		//验证上位机下发数据
		unionSum.words[1]:=modbusdata[650];
		unionSum.words[2]:=modbusdata[649];
		unionSum.words[3]:=modbusdata[648];
		unionSum.words[4]:=modbusdata[647];
		lrSum:=unionSum.lrealValue;
		
		lrSumlocal:=lrFun1_az[10]+lrFun2_az[10]+lrFun3_az[10]+lrFun4_az[10]+lrFun5_az[10]+lrFun6_az[10]
					+lrFun1_el[10]+lrFun2_el[10]+lrFun3_el[10]+lrFun4_el[10]+lrFun5_el[10]+lrFun6_el[10];
		*)
		
		IF NOT bNotFirst THEN
			bCheck := TRUE; // 接收系数完成 开始检测 检测一次
		END_IF
		bNotFirst := TRUE;
	ELSE // 多项式相关变量清零
		bCheck := FALSE;
		bNotFirst := FALSE;
		rNodeTime1_az := 0.0;
		rNodeTime2_az := 0.0;
		rNodeTime3_az := 0.0;
		rNodeTime4_az := 0.0;
		rNodeTime5_az := 0.0;
		rEndTime := 0.0;
		
		FOR i := 0 TO 10 DO
			lrFun1_az[i] := 0;
			lrFun2_az[i] := 0;
			lrFun3_az[i] := 0;
			lrFun4_az[i] := 0;
			lrFun5_az[i] := 0;
			lrFun6_az[i] := 0;
			lrFun3_el[i] := 0;
			lrFun4_el[i] := 0;
		END_FOR
		
		rNodeTime1_el := 0;
		rNodeTime2_el := 0;
		rNodeTime3_el := 0;
		rNodeTime4_el := 0;
		rNodeTime5_el := 0;
		
		FOR i := 0 TO 5 DO
			lrFun1_el[i] := 0;
			lrFun2_el[i] := 0;
			lrFun5_el[i] := 0;
			lrFun6_el[i] := 0;
		END_FOR
	END_IF
	
END_IF

                  
END_PROGRAM

PROGRAM Az_ctrl_1
VAR
    Axis2_Ctrl : Az_Ctrl_FB;
    bRemote2LocalStop : BOOL;
    bLocal2RemoteStop : BOOL;
    Error : INT;
    Axis2Limit_pos : REAL;
    Axis2Limit_Neg : REAL;
    bRTriger : Standard.R_TRIG;
    bFTriger : Standard.F_TRIG;
    Stop2_Count : INT;
    bStop_2 : BOOL;
    rPosModeStepBias : LREAL;
    rPosModeStep : LREAL := 0.005;
    rStepBiasMax : LREAL := 2;
    rStepBias : LREAL;
    rStep : LREAL := 0.002;
    rAuToStepBias : LREAL;
    rAuToStepBiasTemp : LREAL;
    rAutoStep : LREAL := 0.005;
    TbAutoTrigger : Standard.F_TRIG;
    RbAutoTrigger : Standard.R_TRIG;
    rAutoTrackingBiasMax : LREAL := 15;
    rLocalInitPosModeSpeed : REAL;
    rRemoteInitPosModeSpeed : REAL;
    iCountOffAuto : INT;
    iCasePBAutoTrack : INT := 2;
    rKAuToStepBias : LREAL := 0.6; // 对齐2.4
    bVisError : BOOL;
    a : INT;
    agcmaxsearch_tb : agcmaxsearch_pb_1;
    rSearchNextStepTarget_tb : REAL;
    agcmaxsearch_pb : agcmaxsearch_pb_1;
    rElthreshold : REAL := 4.2;
    toN1 : Standard.Ton;
    ttime1 : TIME := T#200mS;
    bstartagcmaxsearch : BOOL;
    rSearchNextStepTarget : REAL;
    rMaxPosTest : REAL;
    iCountSearch : UINT;
    iCountn : UINT;
    bstartSearchAz : BOOL;
    bstartSearchEl : BOOL;
    iCircly : INT := 400;
    rAZSearchThr : REAL := 0.3;
    rElSearchThr : REAL := 0.3;
END_VAR

                    a := 2;
IF GVL.Error_code <> 0 THEN
	bVisError := TRUE;
ELSE
	bVisError := FALSE;
END_IF
(*
//远控轴参量赋值
Axis2Remote.iMode:=Modbus_Slave.iMode_2;
Axis2Remote.rVelCmd:=Modbus_Slave.rVelcmd_2;
Axis2Remote.rPosCmd:=Modbus_Slave.rPosCmd_2;
Axis2Remote.rP:=Modbus_Slave.rP_2;
Axis2Remote.rI:=Modbus_Slave.rI_2;
Axis2Remote.rD:=Modbus_Slave.rD_2;
Axis2Remote.rPIDThre:=Modbus_Slave.rThreshold_2;
Axis2Remote.rAcceleration:=Modbus_Slave.rAcceleration_2;
Axis2Remote.rDeceleration:=Modbus_Slave.rDeceleration_2;
Axis2Remote.rVel_Limit:=Modbus_Slave.rVelLim_2;
*)
// 方位状态写入
Axis2Status.Error := GVL.bAzStsBit3;
Axis2Status.ErrorID := GVL.eAzErrorcode;
Axis2Status.bServo_Enable := GVL.bAzStsBit0 AND GVL.bAzStsBit1 AND GVL.bAzStsBit2;
Axis2Status.bBrake := NOT (GVL.bAzStsBit0 AND GVL.bAzStsBit1 AND GVL.bAzStsBit2);
Axis2Status.Disabled := NOT (GVL.bAzStsBit0 AND GVL.bAzStsBit1 AND GVL.bAzStsBit2);
Axis2Remote.rSoft_limit_Negative:=-275;Axis2Remote.rSoft_limit_Postive:=275;
Axis2Local.rSoft_limit_Negative:=-275;Axis2Local.rSoft_limit_Postive:=275;

//速度的写入
rFctVelReal_2:=DINT_TO_REAL(diAzActVel)/524288.0*360.0;
//位置的写入，方位0对应编码器0，所以实际方位是：-1*编码器值
rFctPosReal_2:=DINT_TO_REAL(diAzActPos)/524288.0*360.0;

//软限位控制
Axis2Limit_pos:=275;
Axis2Limit_Neg:=-275;
IF Axis2Remote.rPosCmd>Axis2Limit_pos THEN
	Axis2Remote.rPosCmd:=275;
ELSIF Axis2Remote.rPosCmd<Axis2Limit_Neg THEN
	 Axis2Remote.rPosCmd:=-275;  
END_IF

IF Axis2Local.rPosCmd>Axis2Limit_pos THEN
	Axis2Local.rPosCmd:=275;
ELSIF Axis2Local.rPosCmd<Axis2Limit_Neg THEN
	 Axis2Local.rPosCmd:=-275;  
END_IF

//停止标志符号判断
IF  ABS(rFctVelReal_2)<0.035 THEN
	Stop2_Count:=Stop2_Count+1;
	IF Stop2_Count>100 THEN
		Stop2_Count:=101;
		bStop_2:=TRUE;;
	END_IF
ELSE
	Stop2_Count:=0;
	bStop_2:=FALSE;
END_IF
Axis2Status.Moving := NOT bStop_2;
//PID使能赋值
IF Axis2Remote.iMode=2 OR Axis2Remote.iMode=4 THEN
	Axis2Remote.bPIDEnable:=TRUE;
ELSE
	Axis2Remote.bPIDEnable:=FALSE;
END_IF

//本远控逻辑保护
//远控切本控逻辑保护
bRTriger(CLK:=GVL.bLocalCtrl);
bFTriger(CLK:=GVL.bLocalCtrl);

IF Axis2Status.bServo_Enable AND (bRTriger.Q ) THEN//如果速度不为0且本控发生切换，则减速停止标识为True
	bRemote2LocalStop:=TRUE;
END_IF
IF bRemote2LocalStop  THEN //若减速停止标识符为True 
	
	IF  bStop_2=TRUE THEN//且电机速度不为0 开始减速 减速完成后下使能，下使能完成后复位标识符复位
		Axis2Local.iMode:=0;
		Axis2Remote.iMode:=0;
		IF Axis2Status.bServo_Enable=FALSE THEN
			bRemote2LocalStop:=FALSE;
		END_IF
	ELSE
		Axis2Local.iMode:=7;
		Axis2Remote.iMode:=7;
	END_IF
END_IF

//本控切远控
IF Axis2Status.bServo_Enable AND (bFTriger.Q ) THEN//如果速度不为0且本控发生切换，则减速停止标识为True
	bLocal2RemoteStop:=TRUE;
END_IF
IF bLocal2RemoteStop  THEN //若减速停止标识符为True 
	
	IF  bStop_2=TRUE THEN//且电机速度不为0 开始减速 减速完成后下使能，下使能完成后复位标识符复位
		Axis2Local.iMode:=0;
		Axis2Remote.iMode:=0;
		IF Axis2Status.bServo_Enable=FALSE THEN
			bLocal2RemoteStop:=FALSE;
		END_IF
	ELSE
		Axis2Remote.iMode:=7;
		Axis2Local.iMode:=7;
	END_IF
END_IF

IF Axis2Remote.iMode=2 THEN
			bstartagcmaxsearch:=Modbus_slave.bSearch;
			IF GVL.Chan1AGC>=(GVL.Chanthreshold-0.1) THEN
					agcmaxsearch_tb(bstart:=bstartagcmaxsearch,rAGCNow:=GVL.Chan1AGC,btrig:=bstartSearchAz,
				rinterPos:=Axis2Remote.rPosCmd,rcurrentpos:=GVL.rFctPosReal_2,
				//rOutStepBias:=0,
				rStepBiasNow:=0,bAutoTracking:=GVL.bStartTrack,bStop:=FALSE,
				rStepBias=>rSearchNextStepTarget_tb,rAGCMaxBias=>rMaxPosTest,bSucess=>);
			ELSE
				bstartagcmaxsearch:=FALSE;
				agcmaxsearch_tb(bstart:=bstartagcmaxsearch,rAGCNow:=GVL.Chan1AGC,btrig:=bstartSearchAz,
				rinterPos:=Axis2Remote.rPosCmd,rcurrentpos:=GVL.rFctPosReal_2,
				//rOutStepBias:=0,
				rStepBiasNow:=0,bAutoTracking:=GVL.bStartTrack,bStop:=FALSE,
				rStepBias=>rSearchNextStepTarget_tb,rAGCMaxBias=>rMaxPosTest,bSucess=>);
			END_IF
			//把rSearchNextStepTarget附加到rPosCmd上
		ELSIF Axis2Remote.iMode=4 AND (GVL.rFctPosReal_1 - 90)>rElthreshold  THEN
			bstartagcmaxsearch:=Modbus_slave.bSearch;
			IF GVL.Chan1AGC>=(GVL.Chanthreshold-0.1) THEN
					agcmaxsearch_pb(bstart:=bstartagcmaxsearch,rAGCNow:=GVL.Chan1AGC,btrig:=bstartSearchAz,
				rinterPos:=RealTimeposcal.rInterAzPos,rcurrentpos:=GVL.rFctPosReal_2,
				//rOutStepBias:=rStepBias,
				rStepBiasNow:=rStepBias,bAutoTracking:=GVL.bStartTrack,bStop:=FALSE,
				rStepBias=>rSearchNextStepTarget,rAGCMaxBias=>rMaxPosTest,bSucess=>);
			ELSE
				bstartagcmaxsearch:=FALSE;
				agcmaxsearch_pb(bstart:=bstartagcmaxsearch,rAGCNow:=GVL.Chan1AGC,btrig:=bstartSearchAz,
				rinterPos:=RealTimeposcal.rInterAzPos,rcurrentpos:=GVL.rFctPosReal_2,
				//rOutStepBias:=rStepBias,
				rStepBiasNow:=rStepBias,bAutoTracking:=GVL.bStartTrack,bStop:=FALSE,
				rStepBias=>rSearchNextStepTarget,rAGCMaxBias=>rMaxPosTest,bSucess=>);
			END_IF
			//把rSearchNextStepTarget附加到Axis2Remote.rPIDCmdPos上
		ELSIF Axis2Remote.iMode =0  OR Axis2Remote.iMode =7 THEN
			bstartagcmaxsearch:=FALSE;
			iCountSearch:=0;
			//rSearchNextStepTarget:=0;
			agcmaxsearch_pb(bstart:=bstartagcmaxsearch,rAGCNow:=GVL.Chan1AGC,btrig:=bstartSearchAz,
			rinterPos:=RealTimeposcal.rInterAzPos,rcurrentpos:=GVL.rFctPosReal_2,
			//rOutStepBias:=rStepBias,
			rStepBiasNow:=rStepBias,bAutoTracking:=GVL.bStartTrack,bStop:=FALSE,
			rStepBias=>rSearchNextStepTarget,rAGCMaxBias=>rMaxPosTest,bSucess=>);
		END_IF
		
(*
//自跟踪
IF GVL.bStartTrack THEN
	Axis2Remote.bStartAutoTrack := TRUE;
	Axis2Remote.rChanU := -AutoTrackingCal.rChanUa;
ELSE
	Axis2Remote.bStartAutoTrack := FALSE;	
	Axis2Remote.rChanU := 0;
END_IF
*)
// 程引模式下自跟踪拉偏
IF GVL.bStartTrack AND Axis2Remote.iMode=4 THEN
	Axis2Remote.bStartAutoTrack := TRUE;
	IF rAuToStepBias > rAutoTrackingBiasMax THEN
		rAuToStepBias := rAutoTrackingBiasMax;
	ELSIF rAuToStepBias < -rAutoTrackingBiasMax THEN
		rAuToStepBias := -rAutoTrackingBiasMax;
	ELSE
		rAuToStepBiasTemp:=(-0.04)*AutoTrackingCal.rDirSenFac*AutoTrackingCal.rChanUa;
		rAuToStepBias:=rAuToStepBias-AutoTrackingCal.rDirSenFac*rKAuToStepBias*AutoTrackingCal.rChanUa/1000.0;
	END_IF
ELSIF NOT GVL.bStartTrack AND Axis2Remote.iMode=4 THEN
	IF 	rAuToStepBias>0 THEN//关闭自跟踪后自跟踪拉偏量逐渐归0
		rAuToStepBias:=rAuToStepBias-rAutoStep;
	ELSIF rAuToStepBias<0 THEN
		rAuToStepBias:=rAuToStepBias+rAutoStep;
	ELSE
		rAuToStepBias:=0;
	END_IF
	
	IF Modbus_Slave.rBias_2>rStepBias THEN
		rStepBias:=rStepBias+rStep;
		IF rStepBias>=Modbus_Slave.rBias_2 THEN
			rStepBias:=Modbus_Slave.rBias_2;
		END_IF
	ELSIF Modbus_Slave.rBias_2<rStepBias THEN
		rStepBias:=rStepBias-rStep;
		IF rStepBias<=Modbus_Slave.rBias_2 THEN
			rStepBias:=Modbus_Slave.rBias_2;
		END_IF
	END_IF
	rAuToStepBiasTemp:=0;
ELSIF GVL.bStartTrack AND Axis2Remote.iMode=2 THEN
	Axis2Remote.bStartAutoTrack := TRUE;
	Axis2Remote.rChanU := -AutoTrackingCal.rChanUa;
ELSE
	Axis2Remote.bStartAutoTrack := FALSE;	
	rAuToStepBias:=0;
	rStepBias:=0;
	rAuToStepBiasTemp:=0;
END_IF

//本控自跟踪
IF GVL.bStartLocalAutoTrack AND Axis2Local.iMode = 4 THEN
	Axis2Local.bStartAutoTrack := TRUE;
	Axis2Local.rChanU := -AutoTrackingCal.rChanUaLocal;
ELSE
	Axis2Local.bStartAutoTrack := FALSE;
END_IF
//拉偏
Axis2Remote.rPIDCmdPos:=RealTimePosCal.rInterAzPos+rStepBias+rAuToStepBias+rSearchNextStepTarget-SECURITYCHECK.AZ_out+rAuToStepBiasTemp;

//限位
IF Axis2Remote.rPIDCmdPos<-275 THEN
	Axis2Remote.rPIDCmdPos:=-275;
ELSIF Axis2Remote.rPIDCmdPos>275 THEN
	Axis2Remote.rPIDCmdPos:=275;
END_IF

Axis2_Ctrl(sLocal:=Axis2Local, sCtrl:=Axis2Remote, sStatus:=Axis2Status, sVisible:=Axis2Visible, rRealPos:=rFctPosReal_2, rPosLimK:=0.34);
	

                  
END_PROGRAM

FUNCTION_BLOCK Az_Ctrl_FB
VAR_INPUT
	sLocal:AxisCrtlStruct;
	sCtrl:AxisCrtlStruct;
	sStatus:AxisStatus;
	sVisible:AxisVisible;
	rRealPos:REAL;
	rPosLimK:REAL;
END_VAR
VAR_OUTPUT
	logicError:INT;
END_VAR
VAR
	VelPID_1:PID;
	VelPID_2:PID;
	VelPID_3:PID;
	vpid1:vpid;
	TON_0:TON;
	bTick:BOOL;
	tr:BOOL;
	icount1:INT := 0;
	icount2:INT := 0;
	icount3:INT := 0;
	bfin1:BOOL;
	bfin2:BOOL;
	istate:INT:=0;
	icount:INT:=0;
END_VAR

                    // 下电时复位控制字bit8
IF sStatus.Disabled OR(NOT sStatus.Moving)THEN
	bAzCtrlBit8 := FALSE;
END_IF

//	错误复位功能
IF GVL.bError_Reset THEN
	sCtrl.iMode:=6;
	sLocal.iMode:=6;
	GVL.Error_code:=0;
END_IF
IF GVL.Error_code =0 THEN
	GVL.bError_Reset:=FALSE;
END_IF

/////////心跳报错清除/////////
IF GVL.eAzErrorcode = 16#8130 AND NOT tr THEN
	GVL.bAzCtrlBit7 := TRUE;
	tr:=TRUE;
	istate:=0;
	icount:=0;
	// 写入下电控制字
	GVL.bAzCtrlBit3 := FALSE;
	GVL.bAzCtrlBit0 := FALSE;
	GVL.bAzCtrlBit1 := FALSE;
	GVL.bAzCtrlBit2 := FALSE;
END_IF
IF tr THEN
	icount1 := icount1 + 1;
END_IF
IF icount1 > 101 THEN
	icount1 := 0;
	tr := FALSE;
	GVL.bAzCtrlBit7 := FALSE;
	bfin1 := TRUE;
END_IF
IF bfin1 THEN
	icount2 := icount2 + 1;
END_IF
IF icount2 > 101 THEN
	bfin1 := FALSE;
	icount2 := 0;
END_IF
/////////////////////////////

IF GVL.Error_code=0 AND GVL.eAzErrorcode = 0 AND NOT GVL.bAzCtrlBit7  AND NOT tr AND NOT bfin1 AND NOT bfin2 THEN
	IF GVL.bLocalCtrl=FALSE THEN //远控
		IF sCtrl.iMode <> 1 THEN
			istate:=0;
			icount:=0;
		END_IF
		CASE sCtrl.iMode OF
			MODES.powerOff: // 下电
				IF NOT sStatus.Disabled THEN
					IF sStatus.Moving THEN // 运动中，先停止运动
						GVL.diAzTargetVel := 0;
						bAzCtrlBit8 := TRUE;
					ELSE
						// 写入下电控制字
						GVL.bAzCtrlBit3 := FALSE;
						GVL.bAzCtrlBit0 := FALSE;
						GVL.bAzCtrlBit1 := FALSE;
						GVL.bAzCtrlBit2 := FALSE;
					END_IF
				END_IF
				
				vpid1(rKpbase:=1, rKibase:=0.01, rKpMax:=1, rKiMax:=0.01, rVelThreshold:=10,rTarget:=sCtrl.rPIDCmdPos,rFeedback:=rRealPos,rPosLimPositive:=sCtrl.rSoft_limit_Postive,
							rPosLimNegitive:=sCtrl.rSoft_limit_Negative,
								bPIDEnable:=sCtrl.bPIDEnable,rVelLim:=sCtrl.rVel_Limit,rKpScale:=0.02,rKiScale:=0.005,rElPos:=GVL.rFctPosReal_1-90,
								iThrehold:=sCtrl.rPIDThre,rPIDOutDir=>sCtrl.rPIDCmdVel);
			MODES.powerOn:  // 上电
				IF sStatus.Disabled THEN
					// 目标速度清零
					GVL.diAzTargetVel := 0;
					IF GVL.siAzMode <> 3 THEN // 上电时模式默认为3，速度模式
						GVL.siAzMode := 3;
					END_IF
					IF siAzMode = 3 THEN
						CASE istate OF
							0:
								GVL.bAzCtrlBit1 := TRUE;
								GVL.bAzCtrlBit2 := TRUE;
								icount := icount + 1;
								IF icount = 20 THEN
									icount:=0;
									istate:=1;
								END_IF
							1:
								GVL.bAzCtrlBit0 := TRUE;
								icount := icount + 1;
								IF icount = 20 THEN
									icount:=0;
									istate:=2;
								END_IF
							2:
								GVL.bAzCtrlBit3 := TRUE;
						END_CASE
					END_IF
				ELSE
					IF sStatus.Moving THEN
						GVL.diAzTargetVel := 0;
						bAzCtrlBit8 := TRUE;
					ELSE
						bAzCtrlBit8 := FALSE;
					END_IF
				END_IF
			MODES.positionMode: // 远控指向模式
				IF NOT sStatus.Disabled THEN
					IF sCtrl.bStartAutoTrack THEN
						//自跟踪模式下，由误差电压直接驱动
						VelPID_1(rTarget:=sCtrl.rChanU + rRealPos,
								rFeedback:=rRealPos,
								rPosLimPositive:=sCtrl.rSoft_limit_Postive,
								rPosLimNegative:=sCtrl.rSoft_limit_Negative,
								rVelLim:=sCtrl.rVel_Limit,
								rKp:=1,//自跟踪PI系数3,0.02
								rKi:=0,
								rKd:=0,
								bPIDEnable:=sCtrl.bPIDEnable,
								iThreshold:= -1,
								rPIDOutput=>sCtrl.rPIDCmdVel);							
					ELSE
						//PID计算速度指令
						VelPID_1(rTarget:=sCtrl.rPosCmd,
							rFeedback:=rRealPos,
							rVelLim:=sCtrl.Pos_Vel,
							rPosLimPositive:=sCtrl.rSoft_limit_Postive,
							rPosLimNegative:=sCtrl.rSoft_limit_Negative,
							rKp:=0.6,//程引PI系数低带：1,0.002  高带：3,0.02
							rKi:=0,
							rKd:=0,
							bPIDEnable:=sCtrl.bPIDEnable,
							iThreshold:=sCtrl.rPIDThre,
							rPIDOutput=>sCtrl.rPIDCmdVel);
					END_IF
					GVL.diAzTargetVel := REAL_TO_DINT(sCtrl.rPIDCmdVel * 524288 / 360);
					GVL.diAzTargetAcc := REAL_TO_UDINT(12 * 524288 / 360);   //加速度
					GVL.diAzTargetDec := REAL_TO_UDINT(12 * 524288 / 360);   //减速度
				END_IF
			MODES.velocityMode://手控速度模式-远控模式
				IF NOT sStatus.Disabled THEN
					IF ABS(sCtrl.rVelCmd) <= sCtrl.rVel_Limit THEN
						GVL.diAzTargetVel := REAL_TO_DINT(sCtrl.rVelCmd * 524288 / 360);
					ELSIF sCtrl.rVelCmd > sCtrl.rVel_Limit THEN
						GVL.diAzTargetVel := REAL_TO_DINT(sCtrl.rVel_Limit * 524288 / 360);
					ELSE
						GVL.diAzTargetVel := REAL_TO_DINT(-sCtrl.rVel_Limit * 524288 / 360);
					END_IF
					GVL.diAzTargetAcc := REAL_TO_UDINT(sCtrl.rAcceleration * 524288 / 360);   //加速度
					GVL.diAzTargetDec := REAL_TO_UDINT(sCtrl.rDeceleration * 524288 / 360);   //减速度
				END_IF
			MODES.programBootMode://PID速度模式-正常模式 程引
				IF NOT sStatus.Disabled THEN
					IF sCtrl.bStartAutoTrack THEN
						(*
						//自跟踪模式下，由误差电压直接驱动
						VelPID_3(rTarget:=sCtrl.rChanU + rRealPos,
								rFeedback:=rRealPos,
								rPosLimPositive:=sCtrl.rSoft_limit_Postive,
								rPosLimNegative:=sCtrl.rSoft_limit_Negative,
								rVelLim:=sCtrl.rVel_Limit,
								rKp:=sCtrl.rP_AutoTrack,//自跟踪PI系数3,0.02
								rKi:=sCtrl.rI_AutoTrack,
								rKd:=sCtrl.rD,
								bPIDEnable:=sCtrl.bPIDEnable,
								iThreshold:= -1,
								rPIDOutput=>sCtrl.rPIDCmdVel);
								*)
						vpid1(rKpbase:=Persistentvars.rAzKpBase, rKibase:=Persistentvars.rAzKiBase, rKpMax:=Persistentvars.rAzKpMax, rKiMax:=Persistentvars.rAzKiMax, rVelThreshold:=Persistentvars.rAzThre,rTarget:=sCtrl.rPIDCmdPos,rFeedback:=rRealPos,rPosLimPositive:=sCtrl.rSoft_limit_Postive,
							rPosLimNegitive:=sCtrl.rSoft_limit_Negative,
								bPIDEnable:=sCtrl.bPIDEnable,rVelLim:=sCtrl.rVel_Limit,rKpScale:=Persistentvars.rAzKpscale,rKiScale:=Persistentvars.rAzKiscale,rElPos:=GVL.rFctPosReal_1-90,
								iThrehold:=sCtrl.rPIDThre,rPIDOutDir=>sCtrl.rPIDCmdVel);							
					ELSE
						//PID计算速度指令
						(*
						VelPID_3(rTarget:=sCtrl.rPIDCmdPos,
							rFeedback:=rRealPos,
							rVelLim:=sCtrl.rVel_Limit,
							rPosLimPositive:=sCtrl.rSoft_limit_Postive,
							rPosLimNegative:=sCtrl.rSoft_limit_Negative,
							rKp:=sCtrl.rP,//程引PI系数地带：1,0.002  高带：3,0.02
							rKi:=sCtrl.rI,
							rKd:=sCtrl.rD,
							bPIDEnable:=sCtrl.bPIDEnable,
							iThreshold:=sCtrl.rPIDThre,
							rPIDOutput=>);
							*)
						vpid1(rKpbase:=Persistentvars.rAzKpBase, rKibase:=Persistentvars.rAzKiBase, rKpMax:=Persistentvars.rAzKpMax, rKiMax:=Persistentvars.rAzKiMax, rVelThreshold:=Persistentvars.rAzThre,rTarget:=sCtrl.rPIDCmdPos,rFeedback:=rRealPos,rPosLimPositive:=sCtrl.rSoft_limit_Postive,
							rPosLimNegitive:=sCtrl.rSoft_limit_Negative,
								bPIDEnable:=sCtrl.bPIDEnable,rVelLim:=sCtrl.rVel_Limit,rKpScale:=Persistentvars.rAzKpscale,rKiScale:=Persistentvars.rAzKiscale,rElPos:=GVL.rFctPosReal_1-90,
								iThrehold:=sCtrl.rPIDThre,rPIDOutDir=>sCtrl.rPIDCmdVel);
						
					END_IF
					GVL.diAzTargetVel := REAL_TO_DINT(sCtrl.rPIDCmdVel * 524288 / 360);
					GVL.diAzTargetAcc := REAL_TO_UDINT(sCtrl.rAcceleration * 524288 / 360);   //加速度
					GVL.diAzTargetDec := REAL_TO_UDINT(sCtrl.rDeceleration * 524288 / 360);   //减速度
				END_IF
			MODES.reset://重置
				IF NOT sStatus.Disabled THEN
					IF sStatus.Moving THEN
						GVL.diAzTargetVel := 0;
						bAzCtrlBit8 := TRUE;
					ELSE
						bAzCtrlBit8 := FALSE;
					END_IF
				END_IF
			MODES.halt://待机
				IF NOT sStatus.Disabled THEN
					IF sStatus.Moving THEN
						GVL.diAzTargetVel := 0;
						bAzCtrlBit8 := TRUE;
					ELSE
						bAzCtrlBit8 := FALSE;
					END_IF
				END_IF
			
		END_CASE
	ELSE // 本控
		IF sLocal.iMode <> 1 THEN
			istate:=0;
			icount:=0;
		END_IF
		CASE sLocal.iMode OF
			MODES.powerOff: // 下电
				IF NOT sStatus.Disabled THEN
					IF sStatus.Moving THEN // 运动中，先停止运动
						GVL.diAzTargetVel := 0;
						bAzCtrlBit8 := TRUE;
					ELSE
						// 写入下电控制字
						GVL.bAzCtrlBit3 := FALSE;
						GVL.bAzCtrlBit0 := FALSE;
						GVL.bAzCtrlBit1 := FALSE;
						GVL.bAzCtrlBit2 := FALSE;
					END_IF
				END_IF
			MODES.powerOn:  // 上电
				IF sStatus.Disabled THEN
					// 目标速度清零
					GVL.diAzTargetVel := 0;
					IF GVL.siAzMode <> 3 THEN // 上电时模式默认为3，速度模式
						GVL.siAzMode := 3;
					END_IF
					IF siAzMode = 3 THEN
						CASE istate OF
							0:
								GVL.bAzCtrlBit1 := TRUE;
								GVL.bAzCtrlBit2 := TRUE;
								icount := icount + 1;
								IF icount = 20 THEN
									icount:=0;
									istate:=1;
								END_IF
							1:
								GVL.bAzCtrlBit0 := TRUE;
								icount := icount + 1;
								IF icount = 20 THEN
									icount:=0;
									istate:=2;
								END_IF
							2:
								GVL.bAzCtrlBit3 := TRUE;
						END_CASE
					END_IF
				ELSE
					IF sStatus.Moving THEN
						GVL.diAzTargetVel := 0;
						bAzCtrlBit8 := TRUE;
					ELSE
						bAzCtrlBit8 := FALSE;
					END_IF
				END_IF
			MODES.velocityMode://手控速度模式-本控模式
				IF NOT sStatus.Disabled THEN
					IF ABS(sLocal.rVelCmd) <= sLocal.rVel_Limit THEN
						GVL.diAzTargetVel := REAL_TO_DINT(sLocal.rVelCmd * 524288 / 360);
					ELSIF sLocal.rVelCmd > sLocal.rVel_Limit THEN
						GVL.diAzTargetVel := REAL_TO_DINT(sLocal.rVel_Limit * 524288 / 360);
					ELSE
						GVL.diAzTargetVel := REAL_TO_DINT(-sLocal.rVel_Limit * 524288 / 360);
					END_IF
					GVL.diAzTargetAcc := REAL_TO_UDINT(sLocal.rAcceleration * 524288 / 360);   //加速度
					GVL.diAzTargetDec := REAL_TO_UDINT(sLocal.rDeceleration * 524288 / 360);   //减速度
				END_IF
			MODES.programBootMode://本控位置模式
				IF NOT sStatus.Disabled THEN
					IF NOT sLocal.bPIDEnable THEN
						GVL.diAzTargetVel := 0;							
					ELSE
						IF NOT slocal.bStartAutoTrack THEN
							//PID计算速度指令
							 VelPID_2(rTarget:=sLocal.rPosCmd,
									 rFeedback:=rRealPos,
									 rPosLimPositive:=sLocal.rSoft_limit_Postive,//软限位
									 rPosLimNegative:=sLocal.rSoft_limit_Negative,
									 rKp:=0.6,
									 rKi:=0,
									 rKd:=0,
									 iThreshold:=sLocal.rPIDThre,
									 bPIDEnable:=sLocal.bPIDEnable,
									 rVelLim:=sLocal.Pos_Vel,
									 rPIDOutput=>sLocal.rPIDCmdVel);//普通PID
						ELSE
							//PID计算速度指令
							 VelPID_2(rTarget:=sLocal.rChanU + rRealPos,
								rFeedback:=rRealPos,
								rPosLimPositive:=sLocal.rSoft_limit_Postive,
								rPosLimNegative:=sLocal.rSoft_limit_Negative,
								rVelLim:=sLocal.rVel_Limit,
								rKp:=1,//自跟踪PI系数3,0.02
								rKi:=0,
								rKd:=0,
								bPIDEnable:=sLocal.bPIDEnable,
								iThreshold:= -1,
								rPIDOutput=>sLocal.rPIDCmdVel);//普通PID
						END_IF
						
					END_IF
					GVL.diAzTargetVel := REAL_TO_DINT(sLocal.rPIDCmdVel * 524288 / 360);
					GVL.diAzTargetAcc := REAL_TO_UDINT(12 * 524288 / 360);   //加速度
					GVL.diAzTargetDec := REAL_TO_UDINT(12 * 524288 / 360);   //减速度
				END_IF
			MODES.reset://重置
			// 是否需要
			MODES.halt://待机
				IF NOT sStatus.Disabled THEN
					IF sStatus.Moving THEN
						GVL.diAzTargetVel := 0;
						bAzCtrlBit8 := TRUE;
					ELSE
						bAzCtrlBit8 := FALSE;
					END_IF
				END_IF
			
		END_CASE
	END_IF
ELSIF GVL.Error_code<>0 AND GVL.eAzErrorcode = 0 AND NOT GVL.bAzCtrlBit7  AND NOT tr AND NOT bfin1 AND NOT bfin2 THEN
	// 出现错误，轴停止运动
	GVL.diAzTargetVel := 0;
	bAzCtrlBit8 := TRUE;
	TON_0(IN:=bAzCtrlBit8,PT:=T#1S,Q=>,ET=>);//判断stop0执行是否超时,若超时强制下电（手动复位）
	IF TON_0.Q THEN
		bTick:=TRUE;
	END_IF
	IF bTick AND sStatus.Moving THEN // 超时强制下电
		// 写入下电控制字
		GVL.bAzCtrlBit3 := FALSE;
		GVL.bAzCtrlBit0 := FALSE;
		GVL.bAzCtrlBit1 := FALSE;
		GVL.bAzCtrlBit2 := FALSE;
	END_IF
END_IF
                  
END_FUNCTION_BLOCK

FUNCTION_BLOCK solvex

VAR_IN_OUT
	M: ARRAY [1..3, 1..3] OF LREAL ; // 定义3x3矩阵M
    G: ARRAY [1..3] OF LREAL ; // 定义3x1数组G
END_VAR
VAR
    
   
	AdjointMatrix: ARRAY [1..3, 1..3] OF REAL; // 用于存储伴随矩阵
	Determinant: REAL; //行列式
    //M_Inverse: ARRAY [1..3, 1..3] OF REAL; //逆矩阵
    i, j, k: INT;
    Temp: REAL;

   

END_VAR

VAR_OUTPUT
	X: ARRAY [1..3] OF REAL; // 用于存储解x
END_VAR

                    
// 计算矩阵的行列式
Determinant := M[1, 1] * (M[2, 2] * M[3, 3] - M[2, 3] * M[3, 2]) -
               M[1, 2] * (M[2, 1] * M[3, 3] - M[2, 3] * M[3, 1]) +
               M[1, 3] * (M[2, 1] * M[3, 2] - M[2, 2] * M[3, 1]);

(*
// 计算3x3矩阵的伴随矩阵
Determinant := M[1, 1] * (M[2, 2] * M[3, 3] - M[2, 3] * M[3, 2]) -
               M[1, 2] * (M[2, 1] * M[3, 3] - M[2, 3] * M[3, 1]) +
               M[1, 3] * (M[2, 1] * M[3, 2] - M[2, 2] * M[3, 1]);

IF ABS(Determinant) > 1.0E-6 THEN
    FOR i := 1 TO 3 DO
        FOR j := 1 TO 3 DO
            AdjointMatrix[i, j] := M[(i MOD 3) + 1, (j MOD 3) + 1] * M[((i + 1) MOD 3) + 1, ((j + 1) MOD 3) + 1] -
                                   M[(i MOD 3) + 1, ((j + 1) MOD 3) + 1] * M[((i + 1) MOD 3) + 1, (j MOD 3) + 1];
        END_FOR
    END_FOR

    FOR i := 1 TO 3 DO
        FOR j := 1 TO 3 DO
            AdjointMatrix[j, i] := AdjointMatrix[i, j];
            AdjointMatrix[i, j] := AdjointMatrix[i, j] / Determinant;
        END_FOR
    END_FOR
END_IF
*)
// 计算3x3矩阵的伴随矩阵
Determinant := M[1, 1] * (M[2, 2] * M[3, 3] - M[2, 3] * M[3, 2]) -
               M[1, 2] * (M[2, 1] * M[3, 3] - M[2, 3] * M[3, 1]) +
               M[1, 3] * (M[2, 1] * M[3, 2] - M[2, 2] * M[3, 1]);

IF ABS(Determinant) > 1.0E-6 THEN
    FOR i := 1 TO 3 DO
        FOR j := 1 TO 3 DO
            AdjointMatrix[j, i] := ((M[(i MOD 3) + 1, (j MOD 3) + 1] * M[((i + 1) MOD 3) + 1, ((j + 1) MOD 3) + 1] -
                                   M[(i MOD 3) + 1, ((j + 1) MOD 3) + 1] * M[((i + 1) MOD 3) + 1, (j MOD 3) + 1]) / Determinant);
        END_FOR
    END_FOR
END_IF

// 计算X = AdjointMatrix * G
FOR i := 1 TO 3 DO
    X[i] := 0.0;
    FOR j := 1 TO 3 DO
        X[i] := X[i] + AdjointMatrix[i, j] * G[j];
    END_FOR
END_FOR




                  
END_FUNCTION_BLOCK

FUNCTION_BLOCK El_Ctrl_FB
VAR_INPUT
	sLocal:AxisCrtlStruct;
	sCtrl:AxisCrtlStruct;
	sStatus:AxisStatus;
	sVisible:AxisVisible;
	rRealPos:REAL;
	rPosLimK:REAL;
END_VAR
VAR_OUTPUT
	logicError:INT;
END_VAR
VAR
	VelPID_1:PID;
	VelPID_2:PID;
	VelPID_3:PID;
	vpid1:vpid;
	TON_0:TON;
	bTick:BOOL;
	tr:BOOL;
	icount1:INT := 0;
	icount2:INT := 0;
	icount3:INT := 0;
	bfin1:BOOL;
	bfin2:BOOL;
	istate:INT:=0;
	icount:INT:=0;
END_VAR

                    // 下电时复位控制字bit8
IF sStatus.Disabled OR (NOT sStatus.Moving) THEN
	bElCtrlBit8 := FALSE;
END_IF

//	错误复位功能
IF GVL.bError_Reset THEN
	sCtrl.iMode:=6;
	sLocal.iMode:=6;
	GVL.Error_code:=0;
END_IF
IF GVL.Error_code =0 THEN
	GVL.bError_Reset:=FALSE;
END_IF

/////////心跳报错清除/////////
IF GVL.eElErrorcode = 16#8130 AND NOT tr THEN
	GVL.bElCtrlBit7 := TRUE;
	tr:=TRUE;
	istate:=0;
	icount:=0;
	// 写入下电控制字
	GVL.bElCtrlBit3 := FALSE;
	GVL.bElCtrlBit0 := FALSE;
	GVL.bElCtrlBit1 := FALSE;
	GVL.bElCtrlBit2 := FALSE;	
END_IF
IF tr THEN
	icount1 := icount1 + 1;
END_IF
IF icount1 > 101 THEN
	icount1 := 0;
	tr := FALSE;
	GVL.bElCtrlBit7 := FALSE;
	bfin1 := TRUE;
END_IF
IF bfin1 THEN
	icount2 := icount2 + 1;
END_IF
IF icount2 > 101 THEN
	bfin1 := FALSE;
	icount2 := 0;
END_IF
//////////////////////////////

IF GVL.Error_code=0 AND GVL.eElErrorcode = 0 AND NOT GVL.bElCtrlBit7  AND NOT tr AND NOT bfin1 AND NOT bfin2 THEN
	IF GVL.bLocalCtrl=FALSE THEN //远控
		IF sCtrl.iMode <> 1 THEN
			istate:=0;
			icount:=0;
		END_IF
		CASE sCtrl.iMode OF
			MODES.powerOff: // 下电
				IF NOT sStatus.Disabled THEN
					IF sStatus.Moving THEN // 运动中，先停止运动
						GVL.diElTargetVel := 0;
						bElCtrlBit8 := TRUE;
					ELSE
						// 写入下电控制字
						GVL.bElCtrlBit3 := FALSE;
						GVL.bElCtrlBit0 := FALSE;
						GVL.bElCtrlBit1 := FALSE;
						GVL.bElCtrlBit2 := FALSE;
					END_IF
				END_IF
				
				vpid1(rKpbase:=1, rKibase:=0.01, rKpMax:=1, rKiMax:=0.01, rVelThreshold:=10,rTarget:=sCtrl.rPIDCmdPos,rFeedback:=rRealPos,rPosLimPositive:=sCtrl.rSoft_limit_Postive,
							rPosLimNegitive:=sCtrl.rSoft_limit_Negative,
								bPIDEnable:=sCtrl.bPIDEnable,rVelLim:=sCtrl.rVel_Limit,rKpScale:=0.02,rKiScale:=0.005,rElPos:=GVL.rFctPosReal_1-90,
								iThrehold:=sCtrl.rPIDThre,rPIDOutDir=>sCtrl.rPIDCmdVel);
			MODES.powerOn:  // 上电
				IF sStatus.Disabled THEN
					// 目标速度清零
					GVL.diElTargetVel := 0;
					IF GVL.siElMode <> 3 THEN // 上电时模式默认为3，速度模式
						GVL.siElMode := 3;
					END_IF
					IF siElMode = 3 THEN
						CASE istate OF
							0:
								GVL.bElCtrlBit1 := TRUE;
								GVL.bElCtrlBit2 := TRUE;
								icount := icount + 1;
								IF icount = 20 THEN
									icount:=0;
									istate:=1;
								END_IF
							1:
								GVL.bElCtrlBit0 := TRUE;
								icount := icount + 1;
								IF icount = 20 THEN
									icount:=0;
									istate:=2;
								END_IF
							2:
								GVL.bElCtrlBit3 := TRUE;
						END_CASE
					END_IF
				ELSE
					IF sStatus.Moving THEN
						GVL.diElTargetVel := 0;
						bElCtrlBit8 := TRUE;
					ELSE
						bElCtrlBit8 := FALSE;
					END_IF
				END_IF
			MODES.positionMode: // 远控指向模式
				IF NOT sStatus.Disabled THEN
					IF sCtrl.bStartAutoTrack THEN
						//自跟踪模式下，由误差电压直接驱动
						VelPID_1(rTarget:=sCtrl.rChanU + rRealPos,
								rFeedback:=rRealPos,
								rPosLimPositive:=sCtrl.rSoft_limit_Postive,
								rPosLimNegative:=sCtrl.rSoft_limit_Negative,
								rVelLim:=sCtrl.rVel_Limit,
								rKp:=1,//自跟踪PI系数3,0.02
								rKi:=0,
								rKd:=0,
								bPIDEnable:=sCtrl.bPIDEnable,
								iThreshold:= -1,
								rPIDOutput=>sCtrl.rPIDCmdVel);							
					ELSE
						//PID计算速度指令
						VelPID_1(rTarget:=sCtrl.rPosCmd,
							rFeedback:=rRealPos,
							rVelLim:=sCtrl.Pos_Vel,
							rPosLimPositive:=sCtrl.rSoft_limit_Postive,
							rPosLimNegative:=sCtrl.rSoft_limit_Negative,
							rKp:=0.7,//程引PI系数地带：1,0.002  高带：3,0.02
							rKi:=0,
							rKd:=0,
							bPIDEnable:=sCtrl.bPIDEnable,
							iThreshold:=sCtrl.rPIDThre,
							rPIDOutput=>sCtrl.rPIDCmdVel);
					END_IF
					GVL.diElTargetVel := REAL_TO_DINT(sCtrl.rPIDCmdVel * 524288 / 360);
					GVL.diElTargetAcc := REAL_TO_UDINT(9 * 524288 / 360);   //加速度
					GVL.diElTargetDec := REAL_TO_UDINT(9 * 524288 / 360);   //减速度
				END_IF
			MODES.velocityMode://手控速度模式-远控模式
				IF NOT sStatus.Disabled THEN
					IF ABS(sCtrl.rVelCmd) <= sCtrl.rVel_Limit THEN
						GVL.diElTargetVel := REAL_TO_DINT(sCtrl.rVelCmd * 524288 / 360);
					ELSIF sCtrl.rVelCmd > sCtrl.rVel_Limit THEN
						GVL.diElTargetVel := REAL_TO_DINT(sCtrl.rVel_Limit * 524288 / 360);
					ELSE
						GVL.diElTargetVel := REAL_TO_DINT(-sCtrl.rVel_Limit * 524288 / 360);
					END_IF
					GVL.diElTargetAcc := REAL_TO_UDINT(sCtrl.rAcceleration * 524288 / 360);   //加速度
					GVL.diElTargetDec := REAL_TO_UDINT(sCtrl.rDeceleration * 524288 / 360);   //减速度
				END_IF
			MODES.programBootMode://PID速度模式-正常模式 程引
				IF NOT sStatus.Disabled THEN
					IF sCtrl.bStartAutoTrack THEN
						(*
						//自跟踪模式下，由误差电压直接驱动
						VelPID_3(rTarget:=sCtrl.rChanU + rRealPos,
								rFeedback:=rRealPos,
								rPosLimPositive:=sCtrl.rSoft_limit_Postive,
								rPosLimNegative:=sCtrl.rSoft_limit_Negative,
								rVelLim:=sCtrl.rVel_Limit,
								rKp:=sCtrl.rP_AutoTrack,//自跟踪PI系数3,0.02
								rKi:=sCtrl.rI_AutoTrack,
								rKd:=sCtrl.rD,
								bPIDEnable:=sCtrl.bPIDEnable,
								iThreshold:= -1,
								rPIDOutput=>sCtrl.rPIDCmdVel);	
								*)
						vpid1(rKpbase:=Persistentvars.rElKpBase, rKibase:=Persistentvars.rElKiBase, rKpMax:=Persistentvars.rElKpMax, rKiMax:=Persistentvars.rElKiMax, rVelThreshold:=Persistentvars.rElThre,rTarget:=sCtrl.rPIDCmdPos,rFeedback:=rRealPos,rPosLimPositive:=sCtrl.rSoft_limit_Postive,
							rPosLimNegitive:=sCtrl.rSoft_limit_Negative,
								bPIDEnable:=sCtrl.bPIDEnable,rVelLim:=sCtrl.rVel_Limit,rKpScale:=Persistentvars.rElKpscale,rKiScale:=Persistentvars.rElKiscale,rElPos:=GVL.rFctPosReal_1-90,
								iThrehold:=sCtrl.rPIDThre,rPIDOutDir=>sCtrl.rPIDCmdVel);						
					ELSE
						//PID计算速度指令
						(*
						VelPID_3(rTarget:=sCtrl.rPIDCmdPos,
							rFeedback:=rRealPos,
							rVelLim:=sCtrl.rVel_Limit,
							rPosLimPositive:=sCtrl.rSoft_limit_Postive,
							rPosLimNegative:=sCtrl.rSoft_limit_Negative,
							rKp:=sCtrl.rP,//程引PI系数地带：1,0.002  高带：3,0.02
							rKi:=sCtrl.rI,
							rKd:=sCtrl.rD,
							bPIDEnable:=sCtrl.bPIDEnable,
							iThreshold:=sCtrl.rPIDThre,
							rPIDOutput=>);
							*)
						vpid1(rKpbase:=Persistentvars.rElKpBase, rKibase:=Persistentvars.rElKiBase, rKpMax:=Persistentvars.rElKpMax, rKiMax:=Persistentvars.rElKiMax, rVelThreshold:=Persistentvars.rElThre,rTarget:=sCtrl.rPIDCmdPos,rFeedback:=rRealPos,rPosLimPositive:=sCtrl.rSoft_limit_Postive,
							rPosLimNegitive:=sCtrl.rSoft_limit_Negative,
								bPIDEnable:=sCtrl.bPIDEnable,rVelLim:=sCtrl.rVel_Limit,rKpScale:=Persistentvars.rElKpscale,rKiScale:=Persistentvars.rElKiscale,rElPos:=GVL.rFctPosReal_1-90,
								iThrehold:=sCtrl.rPIDThre,rPIDOutDir=>sCtrl.rPIDCmdVel);
					END_IF
					GVL.diElTargetVel := REAL_TO_DINT(sCtrl.rPIDCmdVel * 524288 / 360);
					GVL.diElTargetAcc := REAL_TO_UDINT(sCtrl.rAcceleration * 524288 / 360);   //加速度
					GVL.diElTargetDec := REAL_TO_UDINT(sCtrl.rDeceleration * 524288 / 360);   //减速度
				END_IF
			MODES.reset://重置
				IF NOT sStatus.Disabled THEN
					IF sStatus.Moving THEN
						GVL.diElTargetVel := 0;
						bElCtrlBit8 := TRUE;
					ELSE
						bElCtrlBit8 := FALSE;
					END_IF
				END_IF
			MODES.halt://待机
				IF NOT sStatus.Disabled THEN
					IF sStatus.Moving THEN
						GVL.diElTargetVel := 0;
						bElCtrlBit8 := TRUE;
					ELSE
						bElCtrlBit8 := FALSE;
					END_IF
				END_IF
			
		END_CASE
	ELSE // 本控
		IF sLocal.iMode <> 1 THEN
			istate:=0;
			icount:=0;
		END_IF
		CASE sLocal.iMode OF
			MODES.powerOff: // 下电
				IF NOT sStatus.Disabled THEN
					IF sStatus.Moving THEN // 运动中，先停止运动
						GVL.diElTargetVel := 0;
						bElCtrlBit8 := TRUE;
					ELSE
						// 写入下电控制字
						GVL.bElCtrlBit3 := FALSE;
						GVL.bElCtrlBit0 := FALSE;
						GVL.bElCtrlBit1 := FALSE;
						GVL.bElCtrlBit2 := FALSE;
					END_IF
				END_IF
			MODES.powerOn:  // 上电
				IF sStatus.Disabled THEN
					// 目标速度清零
					GVL.diElTargetVel := 0;
					IF GVL.siElMode <> 3 THEN // 上电时模式默认为3，速度模式
						GVL.siElMode := 3;
					END_IF
					IF siElMode = 3 THEN
						
						
						
						CASE istate OF
							0:
								GVL.bElCtrlBit1 := TRUE;
								GVL.bElCtrlBit2 := TRUE;
								icount := icount + 1;
								IF icount = 20 THEN
									icount:=0;
									istate:=1;
								END_IF
							1:
								GVL.bElCtrlBit0 := TRUE;
								icount := icount + 1;
								IF icount = 20 THEN
									icount:=0;
									istate:=2;
								END_IF
							2:
								GVL.bElCtrlBit3 := TRUE;
						END_CASE
					END_IF
				ELSE
					IF sStatus.Moving THEN
						GVL.diElTargetVel := 0;
						bElCtrlBit8 := TRUE;
					ELSE
						bElCtrlBit8 := FALSE;
					END_IF
				END_IF
			MODES.velocityMode://手控速度模式-本控模式
				IF NOT sStatus.Disabled THEN
					IF ABS(sLocal.rVelCmd) <= sLocal.rVel_Limit THEN
						GVL.diElTargetVel := REAL_TO_DINT(sLocal.rVelCmd * 524288 / 360);
					ELSIF sLocal.rVelCmd > sLocal.rVel_Limit THEN
						GVL.diElTargetVel := REAL_TO_DINT(sLocal.rVel_Limit * 524288 / 360);
					ELSE
						GVL.diElTargetVel := REAL_TO_DINT(-sLocal.rVel_Limit * 524288 / 360);
					END_IF
					GVL.diElTargetAcc := REAL_TO_UDINT(sLocal.rAcceleration * 524288 / 360);   //加速度
					GVL.diElTargetDec := REAL_TO_UDINT(sLocal.rDeceleration * 524288 / 360);   //减速度
				END_IF
			MODES.programBootMode://本控位置模式
				IF NOT sStatus.Disabled THEN
					IF NOT sLocal.bPIDEnable THEN
						GVL.diElTargetVel := 0;							
					ELSE
						IF NOT slocal.bStartAutoTrack THEN
							//PID计算速度指令
							 VelPID_2(rTarget:=sLocal.rPosCmd,
									 rFeedback:=rRealPos,
									 rPosLimPositive:=sLocal.rSoft_limit_Postive,//软限位
									 rPosLimNegative:=sLocal.rSoft_limit_Negative,
									 rKp:=0.7,
									 rKi:=0,
									 rKd:=0,
									 iThreshold:=sLocal.rPIDThre,
									 bPIDEnable:=sLocal.bPIDEnable,
									 rVelLim:=sLocal.Pos_Vel,
									 rPIDOutput=>sLocal.rPIDCmdVel);//普通PID
						ELSE
							 VelPID_2(rTarget:=sLocal.rChanU + rRealPos,
								rFeedback:=rRealPos,
								rPosLimPositive:=sLocal.rSoft_limit_Postive,
								rPosLimNegative:=sLocal.rSoft_limit_Negative,
								rVelLim:=sLocal.rVel_Limit,
								rKp:=1,//自跟踪PI系数3,0.02
								rKi:=0,
								rKd:=0,
								bPIDEnable:=sLocal.bPIDEnable,
								iThreshold:= -1,
								rPIDOutput=>sLocal.rPIDCmdVel);
						END_IF
						
					END_IF
					GVL.diElTargetVel := REAL_TO_DINT(sLocal.rPIDCmdVel * 524288 / 360);
					GVL.diElTargetAcc := REAL_TO_UDINT(9 * 524288 / 360);   //加速度
					GVL.diElTargetDec := REAL_TO_UDINT(9 * 524288 / 360);   //减速度
				END_IF
			MODES.reset://重置
			// 是否需要
			MODES.halt://待机
				IF NOT sStatus.Disabled THEN
					IF sStatus.Moving THEN
						GVL.diElTargetVel := 0;
						bElCtrlBit8 := TRUE;
					ELSE
						bElCtrlBit8 := FALSE;
					END_IF
				END_IF
			
		END_CASE
	END_IF
ELSIF GVL.Error_code<>0 AND GVL.eElErrorcode = 0 AND NOT GVL.bElCtrlBit7  AND NOT tr AND NOT bfin1 AND NOT bfin2 THEN
	// 出现错误，轴停止运动
	GVL.diElTargetVel := 0;
	bElCtrlBit8 := TRUE;
	TON_0(IN:=bElCtrlBit8,PT:=T#1S,Q=>,ET=>);//判断stop0执行是否超时,若超时强制下电（手动复位）
	IF TON_0.Q THEN
		bTick:=TRUE;
	END_IF
	IF bTick AND sStatus.Moving THEN // 超时强制下电
		// 写入下电控制字
		GVL.bElCtrlBit3 := FALSE;
		GVL.bElCtrlBit0 := FALSE;
		GVL.bElCtrlBit1 := FALSE;
		GVL.bElCtrlBit2 := FALSE;
	END_IF
END_IF
                  
END_FUNCTION_BLOCK

PROGRAM El_ctrl_1
VAR
    Axis1_Ctrl : El_Ctrl_FB;
    bRemote2LocalStop : BOOL;
    bLocal2RemoteStop : BOOL;
    Error : INT;
    Axis1Limit_pos : REAL;
    Axis1Limit_Neg : REAL;
    bRTriger : Standard.R_TRIG;
    bFTriger : Standard.F_TRIG;
    Stop1_Count : INT;
    bStop_1 : BOOL;
    rPosModeStepBias : LREAL;
    rPosModeStep : LREAL := 0.005;
    rStepBiasMax : LREAL := 2;
    rStepBias : LREAL;
    rStep : LREAL := 0.002;
    rAuToStepBias : LREAL;
    rAuToStepBiasTemp : LREAL;
    rAutoStep : LREAL := 0.01;
    TbAutoTrigger : Standard.F_TRIG;
    RbAutoTrigger : Standard.R_TRIG;
    rAutoTrackingBiasMax : LREAL := 6;
    rLocalInitPosModeSpeed : REAL;
    rRemoteInitPosModeSpeed : REAL;
    iCountOffAuto : INT;
    iCasePBAutoTrack : INT := 2;
    rKAuToStepBias : LREAL := 0.45; // 对齐2.4
    agcmaxsearch_tb : AGCMaxSearch_PB_1;
    rSearchNextStepTarget_tb : REAL;
    agcmaxsearch_pb : AGCMaxSearch_PB_1;
    rElthreshold : REAL := 4.2;
    toN1 : Standard.Ton;
    ttime1 : TIME := T#200mS;
    bstartagcmaxsearch : BOOL;
    rSearchNextStepTarget : REAL;
    rMaxPosTest : REAL;
END_VAR

                    (*
//远控轴参量赋值
Axis1Remote.iMode:=Modbus_Slave.iMode_1;
Axis1Remote.rVelCmd:=Modbus_Slave.rVelcmd_1;
Axis1Remote.rPosCmd:=Modbus_Slave.rPosCmd_1;
Axis1Remote.rP:=Modbus_Slave.rP_1;
Axis1Remote.rI:=Modbus_Slave.rI_1;
Axis1Remote.rD:=Modbus_Slave.rD_1;
Axis1Remote.rPIDThre:=Modbus_Slave.rThreshold_1;
Axis1Remote.rAcceleration:=Modbus_Slave.rAcceleration_1;
Axis1Remote.rDeceleration:=Modbus_Slave.rDeceleration_1;
Axis1Remote.rVel_Limit:=Modbus_Slave.rVelLim_1;
*)
// 方位状态写入
Axis1Status.Error := GVL.bElStsBit3;
Axis1Status.ErrorID := GVL.eElErrorcode;
Axis1Status.bServo_Enable := GVL.bElStsBit0 AND GVL.bElStsBit1 AND GVL.bElStsBit2;
Axis1Status.bBrake := NOT (GVL.bElStsBit0 AND GVL.bElStsBit1 AND GVL.bElStsBit2);
Axis1Status.Disabled := NOT (GVL.bElStsBit0 AND GVL.bElStsBit1 AND GVL.bElStsBit2);
Axis1Remote.rSoft_limit_Negative:=93;Axis1Remote.rSoft_limit_Postive:=180;
Axis1Local.rSoft_limit_Negative:=93;Axis1Local.rSoft_limit_Postive:=180;

//速度的写入
rFctVelReal_1:=DINT_TO_REAL(diElActVel)/524288.0*360.0;
//位置的写入，方位0对应编码器0，所以实际方位是：-1*编码器值
//rFctPosReal_1:=DINT_TO_REAL(diElActPos)/524288.0*360.0 + 5.339;
rFctPosReal_1:=DINT_TO_REAL(diElActPos)/524288.0*360.0 + modbus_slave.lrElOffset;
//软限位控制
Axis1Limit_pos:=180;
Axis1Limit_Neg:=93;
IF Axis1Remote.rPosCmd>Axis1Limit_pos THEN
	Axis1Remote.rPosCmd:=180;
ELSIF Axis1Remote.rPosCmd<Axis1Limit_Neg THEN
	 Axis1Remote.rPosCmd:=93;  
END_IF

IF Axis1Local.rPosCmd>Axis1Limit_pos THEN
	Axis1Local.rPosCmd:=180;
ELSIF Axis1Local.rPosCmd<Axis1Limit_Neg THEN
	 Axis1Local.rPosCmd:=93;  
END_IF

//停止标志符号判断
IF  ABS(rFctVelReal_1)<0.035 THEN
	Stop1_Count:=Stop1_Count+1;
	IF Stop1_Count>100 THEN
		Stop1_Count:=101;
		bStop_1:=TRUE;;
	END_IF
ELSE
	Stop1_Count:=0;
	bStop_1:=FALSE;
END_IF
Axis1Status.Moving := NOT bStop_1;
//PID使能赋值
IF Axis1Remote.iMode=2 OR Axis1Remote.iMode=4 THEN
	Axis1Remote.bPIDEnable:=TRUE;
ELSE
	Axis1Remote.bPIDEnable:=FALSE;
END_IF

//本远控逻辑保护
//远控切本控逻辑保护
bRTriger(CLK:=GVL.bLocalCtrl);
bFTriger(CLK:=GVL.bLocalCtrl);

IF Axis1Status.bServo_Enable AND (bRTriger.Q ) THEN//如果速度不为0且本控发生切换，则减速停止标识为True
	bRemote2LocalStop:=TRUE;
END_IF
IF bRemote2LocalStop  THEN //若减速停止标识符为True 
	
	IF  bStop_1=TRUE THEN//且电机速度不为0 开始减速 减速完成后下使能，下使能完成后复位标识符复位
		Axis1Local.iMode:=0;
		Axis1Remote.iMode:=0;
		IF Axis1Status.bServo_Enable=FALSE THEN
			bRemote2LocalStop:=FALSE;
		END_IF
	ELSE
		Axis1Local.iMode:=7;
		Axis1Remote.iMode:=7;
	END_IF
END_IF

//本控切远控
IF Axis1Status.bServo_Enable AND (bFTriger.Q ) THEN//如果速度不为0且本控发生切换，则减速停止标识为True
	bLocal2RemoteStop:=TRUE;
END_IF
IF bLocal2RemoteStop  THEN //若减速停止标识符为True 
	
	IF  bStop_1=TRUE THEN//且电机速度不为0 开始减速 减速完成后下使能，下使能完成后复位标识符复位
		Axis1Local.iMode:=0;
		Axis1Remote.iMode:=0;
		IF Axis1Status.bServo_Enable=FALSE THEN
			bLocal2RemoteStop:=FALSE;
		END_IF
	ELSE
		Axis1Remote.iMode:=7;
		Axis1Local.iMode:=7;
	END_IF
END_IF
(*
//自跟踪
IF GVL.bStartTrack THEN
	Axis1Remote.bStartAutoTrack := TRUE;
	Axis1Remote.rChanU := AutoTrackingCal.rChanUe;
ELSE
	Axis1Remote.bStartAutoTrack := FALSE;	
	Axis1Remote.rChanU := 0;
END_IF
*)
IF Axis1Remote.iMode=2 THEN
			IF GVL.Chan1AGC>=(GVL.Chanthreshold-0.1) THEN
					agcmaxsearch_pb(bstart:=Az_ctrl_1.agcmaxsearch_tb.bSucess,rAGCNow:=GVL.Chan1AGC,btrig:=Az_ctrl_1.bstartSearchEl,
						rCurrentPos:=rFctPosReal_1,rInterPos:=Axis1Remote.rPosCmd,
				//rOutStepBias:=rStepBias,	
				rStepBiasNow:=rStepBias,bAutoTracking:=GVL.bStartTrack,bStop:=FALSE,
				rStepBias=>rSearchNextStepTarget_tb,rAGCMaxBias=>rMaxPosTest,bSucess=>);
			ELSE
				bstartagcmaxsearch:=FALSE;
				agcmaxsearch_pb(bstart:=Az_ctrl_1.agcmaxsearch_tb.bSucess,rAGCNow:=GVL.Chan1AGC,btrig:=Az_ctrl_1.bstartSearchEl,
				rCurrentPos:=rFctPosReal_1,rInterPos:=Axis1Remote.rPosCmd,
				//rOutStepBias:=rStepBias,
				rStepBiasNow:=rStepBias,bAutoTracking:=GVL.bStartTrack,bStop:=FALSE,
				rStepBias=>rSearchNextStepTarget_tb,rAGCMaxBias=>rMaxPosTest,bSucess=>);
			END_IF
		ELSIF Axis1Remote.iMode=4 AND rFctPosReal_1-90>rElthreshold  THEN
			IF GVL.Chan1AGC>=(GVL.Chanthreshold-0.1) THEN
					agcmaxsearch_pb(bstart:=Az_ctrl_1.agcmaxsearch_pb.bSucess,rAGCNow:=GVL.Chan1AGC,btrig:=Az_ctrl_1.bstartSearchEl,
						rCurrentPos:=rFctPosReal_1,rInterPos:=RealTimePosCal.rInterElPos,
				//rOutStepBias:=rStepBias,	
				rStepBiasNow:=rStepBias,bAutoTracking:=GVL.bStartTrack,bStop:=FALSE,
				rStepBias=>rSearchNextStepTarget,rAGCMaxBias=>rMaxPosTest,bSucess=>);
			ELSE
				bstartagcmaxsearch:=FALSE;
				agcmaxsearch_pb(bstart:=Az_ctrl_1.agcmaxsearch_pb.bSucess,rAGCNow:=GVL.Chan1AGC,btrig:=Az_ctrl_1.bstartSearchEl,
				rCurrentPos:=rFctPosReal_1,rInterPos:=RealTimePosCal.rInterElPos,
				//rOutStepBias:=rStepBias,
				rStepBiasNow:=rStepBias,bAutoTracking:=GVL.bStartTrack,bStop:=FALSE,
				rStepBias=>rSearchNextStepTarget,rAGCMaxBias=>rMaxPosTest,bSucess=>);
			END_IF
			//把rSearchNextStepTarget附加到AzCtrl.rPIDCmdPos上
		ELSIF Axis1Remote.iMode =0  OR Axis1Remote.iMode =7 THEN
			bstartagcmaxsearch:=FALSE;
			//rSearchNextStepTarget:=0;
			agcmaxsearch_pb(bstart:=Az_ctrl_1.agcmaxsearch_pb.bSucess,rAGCNow:=GVL.Chan1AGC,btrig:=Az_ctrl_1.bstartSearchEl,
			rCurrentPos:=rFctPosReal_1,rInterPos:=RealTimePosCal.rInterElPos,	
			//rOutStepBias:=rStepBias,
			rStepBiasNow:=rStepBias,bAutoTracking:=GVL.bStartTrack,bStop:=FALSE,
			rStepBias=>rSearchNextStepTarget,rAGCMaxBias=>rMaxPosTest,bSucess=>);
		END_IF
// 程引模式下自跟踪拉偏
IF GVL.bStartTrack AND Axis1Remote.iMode=4 THEN
	Axis1Remote.bStartAutoTrack := TRUE;
	IF rAuToStepBias > rAutoTrackingBiasMax THEN
		rAuToStepBias := rAutoTrackingBiasMax;
	ELSIF rAuToStepBias < -rAutoTrackingBiasMax THEN
		rAuToStepBias := -rAutoTrackingBiasMax;
	ELSE
		rAuToStepBiasTemp:=0.02*AutoTrackingCal.rDirSenFac*AutoTrackingCal.rChanUe;
		rAuToStepBias:=rAuToStepBias+AutoTrackingCal.rDirSenFac*rKAuToStepBias*AutoTrackingCal.rChanUe/1000.0;
	END_IF
ELSIF NOT GVL.bStartTrack AND Axis1Remote.iMode=4 THEN
	IF 	rAuToStepBias>0 THEN//关闭自跟踪后自跟踪拉偏量逐渐归0
		rAuToStepBias:=rAuToStepBias-rAutoStep;
	ELSIF rAuToStepBias<0 THEN
		rAuToStepBias:=rAuToStepBias+rAutoStep;
	ELSE
		rAuToStepBias:=0;
	END_IF
	
	IF Modbus_Slave.rBias_1>rStepBias THEN
		rStepBias:=rStepBias+rStep;
		IF rStepBias>=Modbus_Slave.rBias_1 THEN
			rStepBias:=Modbus_Slave.rBias_1;
		END_IF
	ELSIF Modbus_Slave.rBias_1<rStepBias THEN
		rStepBias:=rStepBias-rStep;
		IF rStepBias<=Modbus_Slave.rBias_1 THEN
			rStepBias:=Modbus_Slave.rBias_1;
		END_IF
	END_IF
	rAuToStepBiasTemp:=0;
ELSIF GVL.bStartTrack AND Axis1Remote.iMode=2 THEN
	Axis1Remote.bStartAutoTrack := TRUE;
	Axis1Remote.rChanU := AutoTrackingCal.rChanUe;
ELSE
	Axis1Remote.bStartAutoTrack := FALSE;	
	rAuToStepBias:=0;
	rStepBias:=0;
	rAuToStepBiasTemp:=0;
END_IF

//本控自跟踪
IF GVL.bStartLocalAutoTrack AND Axis1Local.iMode = 4 THEN
	Axis1Local.bStartAutoTrack := TRUE;
	Axis1Local.rChanU := AutoTrackingCal.rChanUeLocal;
ELSE
	Axis1Local.bStartAutoTrack := FALSE;
END_IF

//拉偏
Axis1Remote.rPIDCmdPos:=RealTimePosCal.rInterElPos+rStepBias+rAuToStepBias+rSearchNextStepTarget+SECURITYCHECK.el_out+rAuToStepBiasTemp;
//限位
IF Axis1Remote.rPIDCmdPos<93 THEN
	Axis1Remote.rPIDCmdPos:=93;
ELSIF Axis1Remote.rPIDCmdPos>180 THEN
	Axis1Remote.rPIDCmdPos:=180;
END_IF

Axis1_Ctrl(sLocal:=Axis1Local, sCtrl:=Axis1Remote, sStatus:=Axis1Status, sVisible:=Axis1Visible, rRealPos:=rFctPosReal_1, rPosLimK:=0.34);
                  
END_PROGRAM

FUNCTION_BLOCK LinearInter
VAR_INPUT
	tLastTime:ULINT;//上一时间
	rLastPos:REAL;//上一时间位置
	
	tCurTime:ULINT;//当前时间
	rCurPos:REAL;//当前时间位置
	
	tTargetTime:ULINT;//目标时间
END_VAR
VAR_OUTPUT
	rTargetpos:REAL;//目标时间位置
END_VAR
VAR
	iDelCurLastTime:LREAL:=1.0;//	当前与上一个时间差
	iDelTarCurTime:LREAL:=1.0;//目标与当前时间差
	rK:REAL;//方位斜率
END_VAR

                    //tLastTime:=tLastTime/1000000;
//tCurTime:=tCurTime/1000000;
//tTargetTime:=tTargetTime/1000000;
iDelTarCurTime:=ULINT_TO_LREAL(tTargetTime)-ULINT_TO_LREAL(tCurTime); //x1-x
IF (tCurTime-tLastTime)<>0 THEN
	iDelCurLastTime:=ULINT_TO_LREAL(tCurTime)-ULINT_TO_LREAL(tLastTime);  //x-x0
ELSE
	iDelCurLastTime:=1.0;
END_IF

IF iDelTarCurTime<>0 THEN
	rK:=(rCurPos-rLastPos)/(iDelCurLastTime);
ELSE
	rK:=0;
END_IF
rTargetpos:=rCurPos+rK*iDelTarCurTime;  //y1 + ((y1-y0)/(x1-x0))*(x-x1)
                  
END_FUNCTION_BLOCK

FUNCTION_BLOCK three2
VAR_INPUT
	X:ARRAY [1..5] OF LREAL;
	Y:ARRAY [1..5] OF LREAL;
	y0:REAL:=0;
	yn:REAL:=0;//y0,yn表示的是S''(x0)=f''(x0)=y0，S''(xn)=f''(xn)=yn,自然边界即条件值为0
END_VAR

VAR_OUTPUT
	M :ARRAY [1..5] OF LREAL;
	A: ARRAY [1..5,1..5] OF LREAL;
	D: ARRAY[1..3,1..3] OF LREAL;
	g: ARRAY [1..3] OF LREAL;
	h:ARRAY [1..4] OF LREAL;
END_VAR

VAR
	n:INT:=5;
	
	
	ypie:ARRAY [1..5] OF REAL;
	j:INT;
	i:INT;
	u :ARRAY [1..3] OF REAL;
	n_: ARRAY [1..3] OF REAL;
	M_:ARRAY [1..3] OF REAL;
	solve:solvex;

	
	iCounttest: INT;
	
	
	miu :ARRAY [1..4] OF REAL;
END_VAR

                    //此函数为M值求值函数
//D,h,A,g,M输出量分别为系数矩阵D，插值宽度h，差商表A，g值,M值 
n:=5;
//A(:,1)=Y'
A[1,1]:=Y[1];A[2,1]:=Y[2];A[3,1]:=Y[3];A[4,1]:=Y[4];A[5,1]:=Y[5];

//A(:,1)=Y'
FOR j :=2 TO 5 DO
	FOR i:=j TO 5 DO
		A[i,j]:=(A[i,j-1]- A[i-1,j-1])/(X[i]-X[i-j+1]);
	END_FOR
END_FOR


FOR i:=1 TO (n-1) DO
	h[i]:=X[i+1]-X[i];
END_FOR


//h[1]:=X[2]-X[1];h[2]:=X[3]-X[2];h[3]:=X[4]-X[3];h[4]:=X[5]-X[4];



//D[1,1]:=2;D[2,2]:=2;D[3,3]:=2;

FOR i:=1 TO n-2 DO
	D[i,i]:=2; 
	IF i=1 THEN
		g[i]:=(6/(h[i+1]+h[i]))*(A[i+2,2]-A[i+1,2])-h[i]/(h[i]+h[i+1])*y0;
	ELSIF i=(n-2) THEN
		g[i]:=(6/(h[i+1]+h[i]))*(A[i+2,2]-A[i+1,2])-(1-h[i]/(h[i]+h[i+1]))*yn;
	ELSE
		g[i]:=(6/(h[i+1]+h[i]))*(A[i+2,2]-A[i+1,2]);
	END_IF
END_FOR



FOR i:=2 TO (n-2) DO
	u[i]:=h[i]/(h[i]+h[i+1]);
	n_[i-1]:=h[i]/(h[i-1]+h[i]);
	D[i-1,i]:=n_[i-1];
	D[i,i-1]:=u[i];
END_FOR


solve(M:=D,G:=g,X=>M_);
M[1]:=0;M[5]:=0;M[2]:=M_[1];M[3]:=M_[2];M[4]:=M_[3];


                  
END_FUNCTION_BLOCK

FUNCTION_BLOCK threesimple2
VAR_INPUT
	aUTC_TIME:ARRAY [1..5] OF ULINT;  //用于三次样条插值的数据
	aPosCmd :ARRAY [1..5] OF LREAL;//用于三次样条插值的数据
	
	y0:REAL;
	yn:REAL;//y0,yn表示的是S''(x0)=f''(x0)=y0，S''(xn)=f''(xn)=yn,自然边界即条件值为0
	xt:REAL;//所求目标位置
END_VAR
VAR_OUTPUT
	sout:REAL;
	nout:INT;
END_VAR
VAR
	Three:three2;
	X:ARRAY [1..5] OF LREAL;
	Y:ARRAY [1..5] OF LREAL;
	M :ARRAY [1..5] OF LREAL;
	A: ARRAY [1..5,1..5] OF LREAL;
	D: ARRAY[1..3,1..3] OF LREAL;
	g: ARRAY [1..3] OF LREAL;
	h:ARRAY [1..4] OF LREAL;
	
	n:INT:=5;
	
	p1: ARRAY [1..4] OF REAL;
	p2:ARRAY [1..4] OF REAL;
	p3:ARRAY [1..4] OF REAL;
	p4:ARRAY [1..4] OF REAL;
	i:INT;
	
END_VAR

                    FOR i:=1 TO 5 DO
	X[i]:=ULINT_TO_LREAL(aUTC_TIME[i]);
	Y[i]:=aPosCmd[i];
END_FOR


Three(X:=X,Y:=Y,y0:=y0,yn:=yn,D=>D,h=>h,A=>A,g=>g,M=>M);

FOR i:=1 TO (n-1) DO
	p1[i]:=M[i]*(X[i+1]-xt)*(X[i+1]-xt)*(X[i+1]-xt)/(6*h[i]);
	p2[i]:=M[i+1]*(xt-X[i])*(xt-X[i])*(xt-X[i])/(6*h[i]);
	p3[i]:=(A[i,1]-M[i]/6*(h[i])*(h[i]))*(X[i+1]-xt)/h[i];
	p4[i]:=(A[i+1,1]-M[i+1]/6*(h[i])*(h[i]))*(xt-X[i])/h[i];
	
	
END_FOR


FOR i:=1 TO (n-1) DO
	IF (xt<=X[i+1])AND (xt>=X[i]) THEN
		nout:=i;
		sout:=p1[nout]+p2[nout]+p3[nout]+p4[nout]; 
	ELSIF xt>X[5] THEN
		nout:=4;
	ELSIF xt<X[1]THEN
		nout:=1;
	END_IF
END_FOR


//要不要判断插值模块是否有效？
sout:=p1[nout]+p2[nout]+p3[nout]+p4[nout]; 
(*
IF xt>X[5] THEN
	nout:=4;
	sout:=p1[nout]+p2[nout]+p3[nout]+p4[nout]; 
ELSIF xt<X[1] THEN
	nout:=1;
	sout:=p1[nout]+p2[nout]+p3[nout]+p4[nout]; 
END_IF
*)
                  
END_FUNCTION_BLOCK

FUNCTION_BLOCK InterDataProcess
VAR_INPUT
	ulRealTime: ULINT;//实际时间 单位纳秒
	//aOrbitTime: ARRAY [1..5] OF ULINT;//轨道时间数组
	Arr: ARRAY [1..5] OF ULINT:=[9,0,1,5,4]; // 创建一个包含5个整数的数组 轨道时间数组  起点 1970-01-01 0:00:00 单位纳秒
    
END_VAR
VAR_OUTPUT
	MaxVal, MinVal: ULINT;   // 定义最大值、最小值和循环计数器变量
    MaxIndex, MinIndex: INT; // 定义最大值和最小值的索引
	ulInterRealTime : ULINT;//插值使用的时间
END_VAR
VAR
	i,j: INT;
END_VAR

                    //该功能块查找到轨道时间数组内最大最小值以及索引位置
//找出最大最小值
MaxVal := 0; // 初始化最大值
MinVal := 0; // 初始化最小值
MaxIndex := 0; // 初始化最大值的索引
MinIndex := 0; // 初始化最小值的索引

FOR i := 1 TO 5 DO
    IF Arr[i] <> 0 THEN
        IF MaxVal = 0 THEN
            MaxVal := Arr[i];
            MaxIndex := i;
        ELSIF Arr[i] > MaxVal THEN
            MaxVal := Arr[i];
            MaxIndex := i;
        END_IF

        IF MinVal = 0 THEN
            MinVal := Arr[i];
            MinIndex := i;
        ELSIF Arr[i] < MinVal THEN
            MinVal := Arr[i];
            MinIndex := i;
        END_IF
    END_IF
END_FOR

// MaxVal 和 MinVal 包含了最大值和最小值，不考虑值为0的元素
// MaxIndex 和 MinIndex 包含了最大值和最小值的索引


//当前时间和最大最小比较 
IF ulRealTime<MinVal*1000000 THEN //小于插值范围 取最小时间
	//
	ulInterRealTime:=MinVal*1000000; //应该修改插值位置 而不是时间
ELSIF ulRealTime>MaxVal*1000000THEN //大于插值范围 取最大时间
	//
	ulInterRealTime:=MaxVal*1000000;//应该修改插值位置 而不是时间
ELSE
	//如果内部有0 则不插值选取最新的数据
	FOR j:=1 TO 5 DO
		IF (Arr[i]=0) AND (j<5) THEN
			ulInterRealTime:=Arr[5];//应该修改插值位置 而不是时间
			MaxIndex:=5;
			EXIT;
		ELSIF (Arr[i]=0) AND (j=5) THEN
			//没有输入数据 需要报错吗？
		END_IF
	END_FOR
	//
END_IF
                  
END_FUNCTION_BLOCK

FUNCTION_BLOCK threesimple2_1
VAR_INPUT
	XModbusUL:ARRAY [1..10] OF ULINT:=[1,2,3,4,5,6,7,8,9,10];//输入的Modbus时间数组
	XModbus:ARRAY [1..10] OF LREAL;
	YModbus:ARRAY [1..10] OF LREAL;//输入的Modbus位置数组
	y0:REAL;
	yn:REAL;//y0,yn表示的是S''(x0)=f''(x0)=y0，S''(xn)=f''(xn)=yn,自然边界即条件值为0
	xt:LREAL;//所求目标位置
	
	//bResetErr:BOOL;
END_VAR
VAR_OUTPUT
	sout:REAL;
	nout:INT;
	ErrCode:INT;
	
	bSetZero:BOOL;//Modbus序列清零标识符；
END_VAR
VAR
	Three:three2;
	X:ARRAY [1..5] OF LREAL;
	Y:ARRAY [1..5] OF LREAL;
	
	M :ARRAY [1..5] OF LREAL;
	A: ARRAY [1..5,1..5] OF LREAL;
	D: ARRAY[1..3,1..3] OF LREAL;
	g: ARRAY [1..3] OF LREAL;
	h:ARRAY [1..4] OF LREAL;
	
	n:INT:=5;
	
	p1: ARRAY [1..4] OF REAL;
	p2:ARRAY [1..4] OF REAL;
	p3:ARRAY [1..4] OF REAL;
	p4:ARRAY [1..4] OF REAL;
	i:INT;
	ii:INT;//清空序列
	
	j:INT;//寻找差值区间的循环变量
	k:INT;//插值区间
	iCountOutMaxRange:INT;
	iCountOutMinRange:INT;
	nn:INT;//格式转换循环遍历
	mm:INT;//查重遍历；
END_VAR

                    FOR nn:=1 TO 10 DO
	//XModbus[nn]:=ULINT_TO_LREAL(XModbusUL[nn])*1000000/1000.0;
	XModbus[nn]:=ULINT_TO_LREAL(XModbusUL[nn]-XModbusUL[1])+1.0;
END_FOR
	xt:=xt-ULINT_TO_LREAL(XModbusUL[1])+1.0;
IF ErrCode>0 THEN
	ErrCode:=0;
END_IF


FOR mm:=2 TO 8 DO
	IF XModbus[mm] = XModbus[mm + 1] THEN
		// 找到相等的两个数，进行线性插值
		XModbus[mm + 1] := (XModbus[mm] + XModbus[mm + 2]) / 2.0;
	END_IF;
END_FOR
IF XModbus[1] = XModbus[2] THEN
	// 找到相等的两个数，进行线性插值
	XModbus[1] := XModbus[2]-(XModbus[3]-XModbus[2]);
END_IF;
IF XModbus[9] = XModbus[10] THEN
	// 找到相等的两个数，进行线性插值
	XModbus[10] := XModbus[9]+(XModbus[9]-XModbus[8]);
END_IF;

IF ErrCode <> 0 THEN
	iCountOutMaxRange:=0;
	iCountOutMinRange:=0;
END_IF


//在何处清空序列呢
//bSetZero:=FALSE; //默认不清空

IF  XModbus[10]=0 THEN
	//报错
	ErrCode:=107;//序列为空
ELSE
	IF XModbus[10]-XModbus[1]>2000000 THEN
		sout:=YModbus[10];
	ELSE
		IF xt<XModbus[1] THEN
			sout:=YModbus[1];
			//报故障 累计超时报错
			iCountOutMinRange:=iCountOutMinRange+1;
			IF iCountOutMinRange>5000 THEN
				iCountOutMaxRange:=5001;
				//ErrCode:=108;//偏小超时报错
			END_IF
		ELSIF xt>XModbus[10]  THEN
			sout:=YModbus[10];
			//报故障 累计超时报错
			iCountOutMaxRange:=iCountOutMaxRange+1;
			IF iCountOutMaxRange>5000 THEN
				iCountOutMaxRange:=5001;
				//ErrCode:=109;//偏大超时报错
			END_IF
		ELSE //若所求目标位置在Modbus中间
			iCountOutMaxRange:=0;
			iCountOutMinRange:=0;
			//若不满五个点
			IF XModbus[6]=0 THEN
				sout:=XModbus[10];
			ELSE
				//若满五个点
				//寻找当前插值区间
				FOR j:=2 TO 10 DO
					IF xt<XModbus[j] THEN
						k:=j;
						EXIT;
					END_IF
				END_FOR
				
				IF k=2 THEN
					X[1]:=XModbus[k-1];X[2]:=XModbus[k];X[3]:=XModbus[k+1];X[4]:=XModbus[k+2];X[5]:=XModbus[k+3];
					y[1]:=YModbus[k-1];Y[2]:=YModbus[k];Y[3]:=YModbus[k+1];Y[4]:=YModbus[k+2];Y[5]:=YModbus[k+3];
				ELSIF k>2 AND k<=8 THEN
					X[1]:=XModbus[k-2];X[2]:=XModbus[k-1];X[3]:=XModbus[k];X[4]:=XModbus[k+1];X[5]:=XModbus[k+2];
					Y[1]:=YModbus[k-2];Y[2]:=YModbus[k-1];Y[3]:=YModbus[k];Y[4]:=YModbus[k+1];Y[5]:=YModbus[k+2];
				ELSIF k=9 THEN
					X[1]:=XModbus[k-3];X[2]:=XModbus[k-2];X[3]:=XModbus[k-1];X[4]:=XModbus[k];X[5]:=XModbus[k+1];
					Y[1]:=YModbus[k-3];Y[2]:=YModbus[k-2];Y[3]:=YModbus[k-1];Y[4]:=YModbus[k];Y[5]:=YModbus[k+1];
				ELSIF k=10 THEN
					X[1]:=XModbus[k-4];X[2]:=XModbus[k-3];X[3]:=XModbus[k-2];X[4]:=XModbus[k-1];X[5]:=XModbus[k];
					Y[1]:=YModbus[k-4];Y[2]:=YModbus[k-3];Y[3]:=YModbus[k-2];Y[4]:=YModbus[k-1];Y[5]:=YModbus[k];
				END_IF
				
				
				//开始解算
				Three(X:=X,Y:=Y,y0:=y0,yn:=yn,D=>D,h=>h,A=>A,g=>g,M=>M);
				FOR i:=1 TO (n-1) DO
					p1[i]:=M[i]*(X[i+1]-xt)*(X[i+1]-xt)*(X[i+1]-xt)/(6*h[i]);
					p2[i]:=M[i+1]*(xt-X[i])*(xt-X[i])*(xt-X[i])/(6*h[i]);
					p3[i]:=(A[i,1]-M[i]/6*(h[i])*(h[i]))*(X[i+1]-xt)/h[i];
					p4[i]:=(A[i+1,1]-M[i+1]/6*(h[i])*(h[i]))*(xt-X[i])/h[i];
				END_FOR
				FOR i:=1 TO (n-1) DO
					IF (xt<=X[i+1])AND (xt>=X[i]) THEN
						nout:=i;
						sout:=p1[nout]+p2[nout]+p3[nout]+p4[nout]; 
					ELSIF xt>X[5] THEN
						nout:=4;
					ELSIF xt<X[1]THEN
						nout:=1;
					END_IF
				END_FOR
				sout:=p1[nout]+p2[nout]+p3[nout]+p4[nout]; 
				(*
				IF xt>X[5] THEN
					nout:=4;
					sout:=p1[nout]+p2[nout]+p3[nout]+p4[nout]; 
				ELSIF xt<X[1] THEN
					nout:=1;
					sout:=p1[nout]+p2[nout]+p3[nout]+p4[nout]; 
				END_IF
				*)
				END_IF
			END_IF
			
		END_IF

//修正输入量为长度为10的数组

END_IF	
	




                  
END_FUNCTION_BLOCK

PROGRAM SecurityCheck
VAR
    bPrelimit_Positive_1 : BOOL;
    bPrelimit_Negative_1 : BOOL;
    bPrelimit_Positive_2 : BOOL;
    bPrelimit_Negative_2 : BOOL;
    bPrelimit_1 : BOOL;
    bPrelimit_2 : BOOL;
    bFinallimit_1 : BOOL;
    bFinallimit_2 : BOOL;
    AzError : REAL;
    ElError : REAL;
    rELCurrent : REAL;
    rAzCurrent : REAL;
    rTlCurrent : REAL;
    rAz_realpos : REAL;
    rEL_realpos : REAL;
    fbScan : SpiralScan;
    fbScan1 : SpiralScan_1;
    fbScantest : SpiralScan;
    enabletest : BOOL;
    aztest : REAL;
    eltest : REAL;
    enable : BOOL;
    delta : REAL;
    n_steps : REAL;
    agc_sim : REAL;
    lock_sim : BOOL;
    cycle_cnt : INT;
    sim_done : BOOL;
    az_out : REAL;
    el_out : REAL;
    done_out : BOOL;
    bLockSearch : BOOL;
    rSearchThre : REAL;
    rSearchThreTemp : REAL;
    bStartTrackTemp : BOOL;
    RiseEdge : R_TRIG;
    FallEdge : F_TRIG;
    bAcuTrackInhibit : BOOL;
    icountLostLocking : INT;
    bErrorLock : BOOL;
    icountLostLocking1 : INT;
    bType_out : BOOL;
    iconutwait : INT;
    rdelta : REAL := 0.25;         // 螺旋每格边长(°)，4*rdelta=±1°（1°波束）
    rStep : REAL := 12.0;          // 螺旋每格拍数，对齐2.4
    bFinish : BOOL;
    rAzErrorReal : REAL;
    rElErrorReal : REAL;
    rAlpha : REAL;
    icountBaseLock : INT;
    bScanRun : BOOL;
    bScanDoneOnce : BOOL;
    bScanFound : BOOL;
    az_latch : REAL;
    el_latch : REAL;
    bBaseLock : BOOL;
END_VAR

                    
// --- implementation (ST) ---
// =============================================================================
// 段 1: 安全逻辑用位置（与显示用 rFctPosReal 可能差符号/零点）
// =============================================================================
rAz_realpos := -1 * GVL.rFctPosReal_2;
rEl_realpos := GVL.rFctPosReal_1 - 90;

